LIN {X 0,Y 367.091,Z 171.622,A -85,B 0,C 180,E1 -12891.791,E2 -12891.791} C_VEL
LIN {X 0,Y 363.868,Z 162.966,A -85,B 0,C 180,E1 -12892.197,E2 -12892.197} C_VEL
LIN {X 0,Y 361.894,Z 153.404,A -85,B 0,C 180,E1 -12894.844,E2 -12894.844} C_VEL
LIN {X 0,Y 361.85,Z 153.414,A -85,B 0,C 180,E1 -12897.784,E2 -12897.784} C_VEL
LIN {X 0,Y 361.849,Z 153.41,A -85,B 0,C 180,E1 -12901.285,E2 -12901.285} C_VEL
LIN {X 0,Y 361.856,Z 153.408,A -85,B 0,C 180,E1 -12904.28,E2 -12904.28} C_VEL
LIN {X 0,Y 361.861,Z 153.409,A -85,B 0,C 180,E1 -12907.222,E2 -12907.222} C_VEL
LIN {X 0,Y 361.813,Z 153.413,A -85,B 0,C 180,E1 -12910.751,E2 -12910.751} C_VEL
LIN {X 0,Y 361.817,Z 153.412,A -85,B 0,C 180,E1 -12914.368,E2 -12914.368} C_VEL
LIN {X 0,Y 361.831,Z 153.414,A -85,B 0,C 180,E1 -12917.569,E2 -12917.569} C_VEL
LIN {X 0,Y 361.843,Z 153.411,A -85,B 0,C 180,E1 -12921.572,E2 -12921.572} C_VEL
LIN {X 0,Y 361.87,Z 153.407,A -85,B 0,C 180,E1 -12924.656,E2 -12924.656} C_VEL
LIN {X 0,Y 361.836,Z 153.411,A -85,B 0,C 180,E1 -12928.37,E2 -12928.37} C_VEL
LIN {X 0,Y 361.865,Z 153.412,A -85,B 0,C 180,E1 -12930.952,E2 -12930.952} C_VEL
LIN {X 0,Y 361.882,Z 153.409,A -85,B 0,C 180,E1 -12934.706,E2 -12934.706} C_VEL
LIN {X 0,Y 361.888,Z 153.406,A -85,B 0,C 180,E1 -12938.347,E2 -12938.347} C_VEL
LIN {X 0,Y 361.903,Z 153.403,A -85,B 0,C 180,E1 -12942.093,E2 -12942.093} C_VEL
LIN {X 0,Y 361.978,Z 153.394,A -85,B 0,C 180,E1 -12946.113,E2 -12946.113} C_VEL
LIN {X 0,Y 361.997,Z 153.392,A -85,B 0,C 180,E1 -12949.937,E2 -12949.937} C_VEL
LIN {X 0,Y 362.116,Z 153.374,A -85,B 0,C 180,E1 -12953.313,E2 -12953.313} C_VEL
LIN {X 0,Y 362.261,Z 153.359,A -85,B 0,C 180,E1 -12957.776,E2 -12957.776} C_VEL
LIN {X 0,Y 362.17,Z 153.368,A -85,B 0,C 180,E1 -12961.112,E2 -12961.112} C_VEL
LIN {X 0,Y 362.254,Z 153.361,A -85,B 0,C 180,E1 -12962.224,E2 -12962.224} C_VEL
LIN {X 0,Y 362.117,Z 153.375,A -85,B 0,C 180,E1 -12966.687,E2 -12966.687} C_VEL
LIN {X 0,Y 361.99,Z 153.394,A -85,B 0,C 180,E1 -12970.063,E2 -12970.063} C_VEL
LIN {X 0,Y 361.948,Z 153.4,A -85,B 0,C 180,E1 -12973.868,E2 -12973.868} C_VEL
LIN {X 0,Y 361.893,Z 153.405,A -85,B 0,C 180,E1 -12977.903,E2 -12977.903} C_VEL
LIN {X 0,Y 361.851,Z 153.412,A -85,B 0,C 180,E1 -12981.656,E2 -12981.656} C_VEL
LIN {X 0,Y 361.858,Z 153.413,A -85,B 0,C 180,E1 -12985.295,E2 -12985.295} C_VEL
LIN {X 0,Y 361.854,Z 153.412,A -85,B 0,C 180,E1 -12989.074,E2 -12989.074} C_VEL
LIN {X 0,Y 361.846,Z 153.413,A -85,B 0,C 180,E1 -12992.945,E2 -12992.945} C_VEL
LIN {X 0,Y 361.863,Z 153.408,A -85,B 0,C 180,E1 -12995.637,E2 -12995.637} C_VEL
LIN {X 0,Y 361.826,Z 153.417,A -85,B 0,C 180,E1 -12999.018,E2 -12999.018} C_VEL
LIN {X 0,Y 361.831,Z 153.416,A -85,B 0,C 180,E1 -13002.83,E2 -13002.83} C_VEL
LIN {X 0,Y 361.813,Z 153.413,A -85,B 0,C 180,E1 -13005.948,E2 -13005.948} C_VEL
LIN {X 0,Y 361.81,Z 153.414,A -85,B 0,C 180,E1 -13009.25,E2 -13009.25} C_VEL
LIN {X 0,Y 361.864,Z 153.408,A -85,B 0,C 180,E1 -13012.982,E2 -13012.982} C_VEL
LIN {X 0,Y 361.859,Z 153.412,A -85,B 0,C 180,E1 -13016.631,E2 -13016.631} C_VEL
LIN {X 0,Y 361.914,Z 153.447,A -85,B 0,C 180,E1 -13019.747,E2 -13019.747} C_VEL
LIN {X 0,Y 364.405,Z 165.157,A -85,B 0,C 180,E1 -13022.759,E2 -13022.759} C_VEL
LIN {X 0,Y 365.797,Z 172.397,A -85,B 0,C 180,E1 -13024.556,E2 -13024.556} C_VEL
LIN {X 0,Y 365.286,Z 179.494,A -85,B 0,C 180,E1 -13026.169,E2 -13026.169} C_VEL
LIN {X 0,Y 364.51,Z 187.222,A -85,B 0,C 180,E1 -13027.899,E2 -13027.899} C_VEL
LIN {X 0,Y 369.623,Z 218.201,A -85,B 0,C 180,E1 -13028.851,E2 -13028.851} C_VEL
LIN {X 0,Y 370.153,Z 223.288,A -85,B 0,C 180,E1 -13028.986,E2 -13028.986} C_VEL
LIN {X 0,Y 368.915,Z 295.915,A -85,B 0,C 180,E1 -13030.417,E2 -13030.417} C_VEL
LIN {X 0,Y 368.287,Z 309.127,A -85,B 0,C 180,E1 -13030.889,E2 -13030.889} C_VEL
LIN {X 0,Y 367.402,Z 321.258,A -85,B 0,C 180,E1 -13031.529,E2 -13031.529} C_VEL
LIN {X 0,Y 366.327,Z 333.507,A -85,B 0,C 180,E1 -13032.412,E2 -13032.412} C_VEL
LIN {X 0,Y 365.169,Z 345.099,A -85,B 0,C 180,E1 -13033.508,E2 -13033.508} C_VEL
LIN {X 0,Y 364.127,Z 355.365,A -85,B 0,C 180,E1 -13034.729,E2 -13034.729} C_VEL
LIN {X 0,Y 363.187,Z 364.085,A -85,B 0,C 180,E1 -13036.002,E2 -13036.002} C_VEL
LIN {X 0,Y 362.347,Z 371.969,A -85,B 0,C 180,E1 -13037.396,E2 -13037.396} C_VEL
LIN {X 0,Y 361.485,Z 379.671,A -85,B 0,C 180,E1 -13039.072,E2 -13039.072} C_VEL
LIN {X 0,Y 360.873,Z 386.781,A -85,B 0,C 180,E1 -13041.036,E2 -13041.036} C_VEL
LIN {X 0,Y 360.517,Z 391.513,A -85,B 0,C 180,E1 -13042.72,E2 -13042.72} C_VEL
LIN {X 0,Y 360.346,Z 395.131,A -85,B 0,C 180,E1 -13044.403,E2 -13044.403} C_VEL
LIN {X 0,Y 360.359,Z 397,A -85,B 0,C 180,E1 -13045.525,E2 -13045.525} C_VEL
LIN {X 0,Y 360.302,Z 398.399,A -85,B 0,C 180,E1 -13046.645,E2 -13046.645} C_VEL
LIN {X 0,Y 360.37,Z 400.012,A -85,B 0,C 180,E1 -13048.882,E2 -13048.882} C_VEL
LIN {X 0,Y 360.426,Z 400.229,A -85,B 0,C 180,E1 -13049.999,E2 -13049.999} C_VEL
LIN {X 0,Y 360.37,Z 400.007,A -85,B 0,C 180,E1 -13051.117,E2 -13051.117} C_VEL
LIN {X 0,Y 360.302,Z 398.391,A -85,B 0,C 180,E1 -13053.354,E2 -13053.354} C_VEL
LIN {X 0,Y 360.363,Z 396.988,A -85,B 0,C 180,E1 -13054.474,E2 -13054.474} C_VEL
LIN {X 0,Y 360.377,Z 394.412,A -85,B 0,C 180,E1 -13055.96,E2 -13055.96} C_VEL
LIN {X 0,Y 360.649,Z 390.046,A -85,B 0,C 180,E1 -13057.839,E2 -13057.839} C_VEL
LIN {X 0,Y 361.108,Z 383.913,A -85,B 0,C 180,E1 -13059.804,E2 -13059.804} C_VEL
LIN {X 0,Y 361.732,Z 377.218,A -85,B 0,C 180,E1 -13061.486,E2 -13061.486} C_VEL
LIN {X 0,Y 362.697,Z 368.92,A -85,B 0,C 180,E1 -13063.16,E2 -13063.16} C_VEL
LIN {X 0,Y 363.628,Z 360.414,A -85,B 0,C 180,E1 -13064.551,E2 -13064.551} C_VEL
LIN {X 0,Y 364.63,Z 349.903,A -85,B 0,C 180,E1 -13065.941,E2 -13065.941} C_VEL
LIN {X 0,Y 365.85,Z 338.082,A -85,B 0,C 180,E1 -13067.178,E2 -13067.178} C_VEL
LIN {X 0,Y 366.943,Z 326.189,A -85,B 0,C 180,E1 -13068.133,E2 -13068.133} C_VEL
LIN {X 0,Y 367.901,Z 313.816,A -85,B 0,C 180,E1 -13068.877,E2 -13068.877} C_VEL
LIN {X 0,Y 368.686,Z 301.1,A -85,B 0,C 180,E1 -13069.414,E2 -13069.414} C_VEL
LIN {X 0,Y 369.122,Z 287.728,A -85,B 0,C 180,E1 -13069.751,E2 -13069.751} C_VEL
LIN {X 0,Y 369.96,Z 220.882,A -85,B 0,C 180,E1 -13071.059,E2 -13071.059} C_VEL
LIN {X 0,Y 366.012,Z 195.478,A -85,B 0,C 180,E1 -13071.818,E2 -13071.818} C_VEL
LIN {X 0,Y 364.524,Z 187.205,A -85,B 0,C 180,E1 -13072.087,E2 -13072.087} C_VEL
LIN {X 0,Y 365.792,Z 174.22,A -85,B 0,C 180,E1 -13075.003,E2 -13075.003} C_VEL
LIN {X 0,Y 365.348,Z 169.998,A -85,B 0,C 180,E1 -13076.017,E2 -13076.017} C_VEL
LIN {X 0,Y 363.032,Z 158.382,A -85,B 0,C 180,E1 -13078.944,E2 -13078.944} C_VEL
LIN {X 0,Y 361.897,Z 153.408,A -85,B 0,C 180,E1 -13080.253,E2 -13080.253} C_VEL
LIN {X 0,Y 361.85,Z 153.408,A -85,B 0,C 180,E1 -13084.28,E2 -13084.28} C_VEL
LIN {X 0,Y 361.856,Z 153.411,A -85,B 0,C 180,E1 -13087.221,E2 -13087.221} C_VEL
LIN {X 0,Y 361.808,Z 153.414,A -85,B 0,C 180,E1 -13090.75,E2 -13090.75} C_VEL
LIN {X 0,Y 361.809,Z 153.413,A -85,B 0,C 180,E1 -13094.368,E2 -13094.368} C_VEL
LIN {X 0,Y 361.823,Z 153.414,A -85,B 0,C 180,E1 -13097.568,E2 -13097.568} C_VEL
LIN {X 0,Y 361.837,Z 153.411,A -85,B 0,C 180,E1 -13101.571,E2 -13101.571} C_VEL
LIN {X 0,Y 361.863,Z 153.41,A -85,B 0,C 180,E1 -13104.656,E2 -13104.656} C_VEL
LIN {X 0,Y 361.83,Z 153.412,A -85,B 0,C 180,E1 -13108.37,E2 -13108.37} C_VEL
LIN {X 0,Y 361.859,Z 153.411,A -85,B 0,C 180,E1 -13110.951,E2 -13110.951} C_VEL
LIN {X 0,Y 361.853,Z 153.414,A -85,B 0,C 180,E1 -13114.704,E2 -13114.704} C_VEL
LIN {X 0,Y 361.845,Z 153.412,A -85,B 0,C 180,E1 -13118.344,E2 -13118.344} C_VEL
LIN {X 0,Y 361.896,Z 153.405,A -85,B 0,C 180,E1 -13122.092,E2 -13122.092} C_VEL
LIN {X 0,Y 361.97,Z 153.397,A -85,B 0,C 180,E1 -13126.113,E2 -13126.113} C_VEL
LIN {X 0,Y 361.985,Z 153.394,A -85,B 0,C 180,E1 -13129.937,E2 -13129.937} C_VEL
LIN {X 0,Y 362.108,Z 153.376,A -85,B 0,C 180,E1 -13133.313,E2 -13133.313} C_VEL
LIN {X 0,Y 362.248,Z 153.362,A -85,B 0,C 180,E1 -13137.776,E2 -13137.776} C_VEL
LIN {X 0,Y 362.163,Z 153.369,A -85,B 0,C 180,E1 -13141.112,E2 -13141.112} C_VEL
LIN {X 0,Y 362.254,Z 153.361,A -85,B 0,C 180,E1 -13142.224,E2 -13142.224} C_VEL
LIN {X 0,Y 362.112,Z 153.375,A -85,B 0,C 180,E1 -13146.687,E2 -13146.687} C_VEL
LIN {X 0,Y 361.99,Z 153.393,A -85,B 0,C 180,E1 -13150.063,E2 -13150.063} C_VEL
LIN {X 0,Y 361.971,Z 153.396,A -85,B 0,C 180,E1 -13153.887,E2 -13153.887} C_VEL
LIN {X 0,Y 361.879,Z 153.405,A -85,B 0,C 180,E1 -13158.104,E2 -13158.104} C_VEL
LIN {X 0,Y 361.881,Z 153.407,A -85,B 0,C 180,E1 -13161.654,E2 -13161.654} C_VEL
LIN {X 0,Y 361.854,Z 153.413,A -85,B 0,C 180,E1 -13165.296,E2 -13165.296} C_VEL
LIN {X 0,Y 361.848,Z 153.414,A -85,B 0,C 180,E1 -13169.074,E2 -13169.074} C_VEL
LIN {X 0,Y 361.841,Z 153.414,A -85,B 0,C 180,E1 -13172.946,E2 -13172.946} C_VEL
LIN {X 0,Y 361.858,Z 153.408,A -85,B 0,C 180,E1 -13175.638,E2 -13175.638} C_VEL
LIN {X 0,Y 361.821,Z 153.416,A -85,B 0,C 180,E1 -13179.019,E2 -13179.019} C_VEL
LIN {X 0,Y 361.828,Z 153.417,A -85,B 0,C 180,E1 -13182.83,E2 -13182.83} C_VEL
LIN {X 0,Y 361.813,Z 153.413,A -85,B 0,C 180,E1 -13185.948,E2 -13185.948} C_VEL
LIN {X 0,Y 361.826,Z 153.412,A -85,B 0,C 180,E1 -13189.247,E2 -13189.247} C_VEL
LIN {X 0,Y 361.862,Z 153.408,A -85,B 0,C 180,E1 -13192.983,E2 -13192.983} C_VEL
LIN {X 0,Y 361.857,Z 153.411,A -85,B 0,C 180,E1 -13196.632,E2 -13196.632} C_VEL
LIN {X 0,Y 361.863,Z 153.407,A -85,B 0,C 180,E1 -13199.672,E2 -13199.672} C_VEL
LIN {X 0,Y 361.864,Z 153.406,A -85,B 0,C 180,E1 -13203.469,E2 -13203.469} C_VEL
LIN {X 0,Y 361.905,Z 153.596,A -85,B 0,C 180,E1 -13205.322,E2 -13205.322} C_VEL
LIN {X 0,Y 363.891,Z 162.985,A -85,B 0,C 180,E1 -13207.917,E2 -13207.917} C_VEL
LIN {X 0,Y 367.735,Z 173.936,A -85,B 0,C 180,E1 -13208.403,E2 -13208.403} C_VEL
LIN {X 0,Y 370.621,Z 188.653,A -85,B 0,C 180,E1 -13208.883,E2 -13208.883} C_VEL
LIN {X 0,Y 369.412,Z 265.31,A -85,B 0,C 180,E1 -13210.373,E2 -13210.373} C_VEL
LIN {X 0,Y 369.011,Z 278.206,A -85,B 0,C 180,E1 -13210.749,E2 -13210.749} C_VEL
LIN {X 0,Y 368.333,Z 291.445,A -85,B 0,C 180,E1 -13211.362,E2 -13211.362} C_VEL
LIN {X 0,Y 367.455,Z 303.827,A -85,B 0,C 180,E1 -13212.181,E2 -13212.181} C_VEL
LIN {X 0,Y 366.505,Z 314.918,A -85,B 0,C 180,E1 -13213.141,E2 -13213.141} C_VEL
LIN {X 0,Y 365.734,Z 324.837,A -85,B 0,C 180,E1 -13214.225,E2 -13214.225} C_VEL
LIN {X 0,Y 364.652,Z 334.372,A -85,B 0,C 180,E1 -13215.491,E2 -13215.491} C_VEL
LIN {X 0,Y 363.638,Z 342.859,A -85,B 0,C 180,E1 -13216.875,E2 -13216.875} C_VEL
LIN {X 0,Y 362.729,Z 351.099,A -85,B 0,C 180,E1 -13218.546,E2 -13218.546} C_VEL
LIN {X 0,Y 362.057,Z 356.737,A -85,B 0,C 180,E1 -13219.939,E2 -13219.939} C_VEL
LIN {X 0,Y 361.4,Z 362.232,A -85,B 0,C 180,E1 -13221.614,E2 -13221.614} C_VEL
LIN {X 0,Y 361.035,Z 366.54,A -85,B 0,C 180,E1 -13223.293,E2 -13223.293} C_VEL
LIN {X 0,Y 360.844,Z 368.819,A -85,B 0,C 180,E1 -13224.412,E2 -13224.412} C_VEL
LIN {X 0,Y 360.627,Z 370.676,A -85,B 0,C 180,E1 -13225.53,E2 -13225.53} C_VEL
LIN {X 0,Y 360.515,Z 372.072,A -85,B 0,C 180,E1 -13226.648,E2 -13226.648} C_VEL
LIN {X 0,Y 360.424,Z 373.675,A -85,B 0,C 180,E1 -13228.883,E2 -13228.883} C_VEL
LIN {X 0,Y 360.429,Z 373.906,A -85,B 0,C 180,E1 -13230.001,E2 -13230.001} C_VEL
LIN {X 0,Y 360.424,Z 373.718,A -85,B 0,C 180,E1 -13231.118,E2 -13231.118} C_VEL
LIN {X 0,Y 360.51,Z 372.171,A -85,B 0,C 180,E1 -13233.353,E2 -13233.353} C_VEL
LIN {X 0,Y 360.619,Z 370.818,A -85,B 0,C 180,E1 -13234.472,E2 -13234.472} C_VEL
LIN {X 0,Y 360.934,Z 367.955,A -85,B 0,C 180,E1 -13236.148,E2 -13236.148} C_VEL
LIN {X 0,Y 361.212,Z 364.08,A -85,B 0,C 180,E1 -13237.828,E2 -13237.828} C_VEL
LIN {X 0,Y 361.778,Z 359.072,A -85,B 0,C 180,E1 -13239.505,E2 -13239.505} C_VEL
LIN {X 0,Y 362.531,Z 352.766,A -85,B 0,C 180,E1 -13241.179,E2 -13241.179} C_VEL
LIN {X 0,Y 363.433,Z 344.872,A -85,B 0,C 180,E1 -13242.85,E2 -13242.85} C_VEL
LIN {X 0,Y 364.45,Z 336.819,A -85,B 0,C 180,E1 -13244.234,E2 -13244.234} C_VEL
LIN {X 0,Y 365.523,Z 326.991,A -85,B 0,C 180,E1 -13245.616,E2 -13245.616} C_VEL
LIN {X 0,Y 366.352,Z 317.324,A -85,B 0,C 180,E1 -13246.724,E2 -13246.724} C_VEL
LIN {X 0,Y 367.287,Z 306.852,A -85,B 0,C 180,E1 -13247.684,E2 -13247.684} C_VEL
LIN {X 0,Y 368.181,Z 294.238,A -85,B 0,C 180,E1 -13248.575,E2 -13248.575} C_VEL
LIN {X 0,Y 368.908,Z 281.603,A -85,B 0,C 180,E1 -13249.222,E2 -13249.222} C_VEL
LIN {X 0,Y 369.266,Z 273.016,A -85,B 0,C 180,E1 -13249.53,E2 -13249.53} C_VEL
LIN {X 0,Y 368.777,Z 267.258,A -85,B 0,C 180,E1 -13249.725,E2 -13249.725} C_VEL
LIN {X 0,Y 363.714,Z 248.579,A -85,B 0,C 180,E1 -13250.412,E2 -13250.412} C_VEL
LIN {X 0,Y 363.144,Z 242.768,A -85,B 0,C 180,E1 -13250.561,E2 -13250.561} C_VEL
LIN {X 0,Y 363.993,Z 188.874,A -85,B 0,C 180,E1 -13251.629,E2 -13251.629} C_VEL
LIN {X 0,Y 360.675,Z 173.698,A -85,B 0,C 180,E1 -13252.16,E2 -13252.16} C_VEL
LIN {X 0,Y 356.72,Z 163.234,A -85,B 0,C 180,E1 -13252.667,E2 -13252.667} C_VEL
LIN {X 0,Y 354.855,Z 154.281,A -85,B 0,C 180,E1 -13255.202,E2 -13255.202} C_VEL
LIN {X 0,Y 354.804,Z 154.288,A -85,B 0,C 180,E1 -13258.385,E2 -13258.385} C_VEL
LIN {X 0,Y 354.789,Z 154.289,A -85,B 0,C 180,E1 -13262.333,E2 -13262.333} C_VEL
LIN {X 0,Y 354.823,Z 154.289,A -85,B 0,C 180,E1 -13265.699,E2 -13265.699} C_VEL
LIN {X 0,Y 354.769,Z 154.295,A -85,B 0,C 180,E1 -13269.412,E2 -13269.412} C_VEL
LIN {X 0,Y 354.786,Z 154.289,A -85,B 0,C 180,E1 -13272.867,E2 -13272.867} C_VEL
LIN {X 0,Y 354.767,Z 154.29,A -85,B 0,C 180,E1 -13276.103,E2 -13276.103} C_VEL
LIN {X 0,Y 354.766,Z 154.296,A -85,B 0,C 180,E1 -13279.176,E2 -13279.176} C_VEL
LIN {X 0,Y 354.799,Z 154.287,A -85,B 0,C 180,E1 -13282.404,E2 -13282.404} C_VEL
LIN {X 0,Y 354.808,Z 154.29,A -85,B 0,C 180,E1 -13284.94,E2 -13284.94} C_VEL
LIN {X 0,Y 354.792,Z 154.288,A -85,B 0,C 180,E1 -13288.405,E2 -13288.405} C_VEL
LIN {X 0,Y 354.799,Z 154.286,A -85,B 0,C 180,E1 -13291.614,E2 -13291.614} C_VEL
LIN {X 0,Y 354.834,Z 154.282,A -85,B 0,C 180,E1 -13295.657,E2 -13295.657} C_VEL
LIN {X 0,Y 354.834,Z 154.284,A -85,B 0,C 180,E1 -13299.113,E2 -13299.113} C_VEL
LIN {X 0,Y 354.85,Z 154.284,A -85,B 0,C 180,E1 -13302.717,E2 -13302.717} C_VEL
LIN {X 0,Y 354.938,Z 154.272,A -85,B 0,C 180,E1 -13306.254,E2 -13306.254} C_VEL
LIN {X 0,Y 354.953,Z 154.268,A -85,B 0,C 180,E1 -13309.735,E2 -13309.735} C_VEL
LIN {X 0,Y 355.082,Z 154.25,A -85,B 0,C 180,E1 -13313.18,E2 -13313.18} C_VEL
LIN {X 0,Y 355.223,Z 154.236,A -85,B 0,C 180,E1 -13317.732,E2 -13317.732} C_VEL
LIN {X 0,Y 355.142,Z 154.242,A -85,B 0,C 180,E1 -13321.134,E2 -13321.134} C_VEL
LIN {X 0,Y 355.216,Z 154.237,A -85,B 0,C 180,E1 -13322.268,E2 -13322.268} C_VEL
LIN {X 0,Y 355.083,Z 154.251,A -85,B 0,C 180,E1 -13326.82,E2 -13326.82} C_VEL
LIN {X 0,Y 354.946,Z 154.269,A -85,B 0,C 180,E1 -13330.265,E2 -13330.265} C_VEL
LIN {X 0,Y 354.89,Z 154.278,A -85,B 0,C 180,E1 -13333.985,E2 -13333.985} C_VEL
LIN {X 0,Y 354.833,Z 154.283,A -85,B 0,C 180,E1 -13338.065,E2 -13338.065} C_VEL
LIN {X 0,Y 354.803,Z 154.286,A -85,B 0,C 180,E1 -13342.108,E2 -13342.108} C_VEL
LIN {X 0,Y 354.797,Z 154.288,A -85,B 0,C 180,E1 -13345.835,E2 -13345.835} C_VEL
LIN {X 0,Y 354.791,Z 154.289,A -85,B 0,C 180,E1 -13349.684,E2 -13349.684} C_VEL
LIN {X 0,Y 354.785,Z 154.288,A -85,B 0,C 180,E1 -13352.334,E2 -13352.334} C_VEL
LIN {X 0,Y 354.817,Z 154.285,A -85,B 0,C 180,E1 -13355.698,E2 -13355.698} C_VEL
LIN {X 0,Y 354.768,Z 154.292,A -85,B 0,C 180,E1 -13359.413,E2 -13359.413} C_VEL
LIN {X 0,Y 354.784,Z 154.295,A -85,B 0,C 180,E1 -13362.866,E2 -13362.866} C_VEL
LIN {X 0,Y 354.762,Z 154.292,A -85,B 0,C 180,E1 -13366.103,E2 -13366.103} C_VEL
LIN {X 0,Y 354.763,Z 154.292,A -85,B 0,C 180,E1 -13369.176,E2 -13369.176} C_VEL
LIN {X 0,Y 354.801,Z 154.29,A -85,B 0,C 180,E1 -13372.404,E2 -13372.404} C_VEL
LIN {X 0,Y 354.812,Z 154.288,A -85,B 0,C 180,E1 -13374.941,E2 -13374.941} C_VEL
LIN {X 0,Y 354.794,Z 154.293,A -85,B 0,C 180,E1 -13378.405,E2 -13378.405} C_VEL
LIN {X 0,Y 354.862,Z 154.356,A -85,B 0,C 180,E1 -13379.379,E2 -13379.379} C_VEL
LIN {X 0,Y 357.269,Z 165.329,A -85,B 0,C 180,E1 -13382.278,E2 -13382.278} C_VEL
LIN {X 0,Y 358.884,Z 174.019,A -85,B 0,C 180,E1 -13384.48,E2 -13384.48} C_VEL
LIN {X 0,Y 358.14,Z 183.133,A -85,B 0,C 180,E1 -13386.585,E2 -13386.585} C_VEL
LIN {X 0,Y 357.664,Z 186.937,A -85,B 0,C 180,E1 -13387.449,E2 -13387.449} C_VEL
LIN {X 0,Y 362.658,Z 216.507,A -85,B 0,C 180,E1 -13388.395,E2 -13388.395} C_VEL
LIN {X 0,Y 363.534,Z 223.627,A -85,B 0,C 180,E1 -13388.597,E2 -13388.597} C_VEL
LIN {X 0,Y 362.248,Z 295.669,A -85,B 0,C 180,E1 -13390.041,E2 -13390.041} C_VEL
LIN {X 0,Y 361.592,Z 308.877,A -85,B 0,C 180,E1 -13390.521,E2 -13390.521} C_VEL
LIN {X 0,Y 360.677,Z 321.006,A -85,B 0,C 180,E1 -13391.172,E2 -13391.172} C_VEL
LIN {X 0,Y 359.573,Z 333.252,A -85,B 0,C 180,E1 -13392.071,E2 -13392.071} C_VEL
LIN {X 0,Y 358.335,Z 344.842,A -85,B 0,C 180,E1 -13393.184,E2 -13393.184} C_VEL
LIN {X 0,Y 357.18,Z 355.873,A -85,B 0,C 180,E1 -13394.53,E2 -13394.53} C_VEL
LIN {X 0,Y 356.091,Z 365.505,A -85,B 0,C 180,E1 -13396.008,E2 -13396.008} C_VEL
LIN {X 0,Y 355.061,Z 374.452,A -85,B 0,C 180,E1 -13397.714,E2 -13397.714} C_VEL
LIN {X 0,Y 354.286,Z 381.656,A -85,B 0,C 180,E1 -13399.426,E2 -13399.426} C_VEL
LIN {X 0,Y 353.691,Z 388.222,A -85,B 0,C 180,E1 -13401.429,E2 -13401.429} C_VEL
LIN {X 0,Y 353.397,Z 392.569,A -85,B 0,C 180,E1 -13403.147,E2 -13403.147} C_VEL
LIN {X 0,Y 353.282,Z 394.873,A -85,B 0,C 180,E1 -13404.291,E2 -13404.291} C_VEL
LIN {X 0,Y 353.269,Z 396.741,A -85,B 0,C 180,E1 -13405.435,E2 -13405.435} C_VEL
LIN {X 0,Y 353.223,Z 398.141,A -85,B 0,C 180,E1 -13406.577,E2 -13406.577} C_VEL
LIN {X 0,Y 353.271,Z 399.753,A -85,B 0,C 180,E1 -13408.859,E2 -13408.859} C_VEL
LIN {X 0,Y 353.331,Z 399.97,A -85,B 0,C 180,E1 -13409.999,E2 -13409.999} C_VEL
LIN {X 0,Y 353.271,Z 399.748,A -85,B 0,C 180,E1 -13411.139,E2 -13411.139} C_VEL
LIN {X 0,Y 353.224,Z 398.132,A -85,B 0,C 180,E1 -13413.421,E2 -13413.421} C_VEL
LIN {X 0,Y 353.274,Z 396.728,A -85,B 0,C 180,E1 -13414.563,E2 -13414.563} C_VEL
LIN {X 0,Y 353.275,Z 394.483,A -85,B 0,C 180,E1 -13415.904,E2 -13415.904} C_VEL
LIN {X 0,Y 353.574,Z 389.784,A -85,B 0,C 180,E1 -13417.997,E2 -13417.997} C_VEL
LIN {X 0,Y 354.073,Z 383.651,A -85,B 0,C 180,E1 -13420.001,E2 -13420.001} C_VEL
LIN {X 0,Y 354.719,Z 376.955,A -85,B 0,C 180,E1 -13421.716,E2 -13421.716} C_VEL
LIN {X 0,Y 355.754,Z 368.658,A -85,B 0,C 180,E1 -13423.421,E2 -13423.421} C_VEL
LIN {X 0,Y 356.746,Z 360.152,A -85,B 0,C 180,E1 -13424.838,E2 -13424.838} C_VEL
LIN {X 0,Y 357.763,Z 349.639,A -85,B 0,C 180,E1 -13426.255,E2 -13426.255} C_VEL
LIN {X 0,Y 359.054,Z 337.818,A -85,B 0,C 180,E1 -13427.513,E2 -13427.513} C_VEL
LIN {X 0,Y 360.175,Z 325.923,A -85,B 0,C 180,E1 -13428.486,E2 -13428.486} C_VEL
LIN {X 0,Y 361.195,Z 313.549,A -85,B 0,C 180,E1 -13429.241,E2 -13429.241} C_VEL
LIN {X 0,Y 362.001,Z 300.83,A -85,B 0,C 180,E1 -13429.787,E2 -13429.787} C_VEL
LIN {X 0,Y 362.456,Z 287.449,A -85,B 0,C 180,E1 -13430.13,E2 -13430.13} C_VEL
LIN {X 0,Y 363.351,Z 221.934,A -85,B 0,C 180,E1 -13431.433,E2 -13431.433} C_VEL
LIN {X 0,Y 359.5,Z 196.978,A -85,B 0,C 180,E1 -13432.197,E2 -13432.197} C_VEL
LIN {X 0,Y 357.695,Z 186.921,A -85,B 0,C 180,E1 -13432.536,E2 -13432.536} C_VEL
LIN {X 0,Y 358.877,Z 175.254,A -85,B 0,C 180,E1 -13435.209,E2 -13435.209} C_VEL
LIN {X 0,Y 358.144,Z 169.993,A -85,B 0,C 180,E1 -13436.514,E2 -13436.514} C_VEL
LIN {X 0,Y 355.842,Z 158.873,A -85,B 0,C 180,E1 -13439.394,E2 -13439.394} C_VEL
LIN {X 0,Y 354.831,Z 154.288,A -85,B 0,C 180,E1 -13440.664,E2 -13440.664} C_VEL
LIN {X 0,Y 354.803,Z 154.29,A -85,B 0,C 180,E1 -13443.701,E2 -13443.701} C_VEL
LIN {X 0,Y 354.791,Z 154.287,A -85,B 0,C 180,E1 -13446.459,E2 -13446.459} C_VEL
LIN {X 0,Y 354.764,Z 154.296,A -85,B 0,C 180,E1 -13449.411,E2 -13449.411} C_VEL
LIN {X 0,Y 354.78,Z 154.291,A -85,B 0,C 180,E1 -13452.866,E2 -13452.866} C_VEL
LIN {X 0,Y 354.757,Z 154.292,A -85,B 0,C 180,E1 -13456.102,E2 -13456.102} C_VEL
LIN {X 0,Y 354.76,Z 154.297,A -85,B 0,C 180,E1 -13459.175,E2 -13459.175} C_VEL
LIN {X 0,Y 354.793,Z 154.288,A -85,B 0,C 180,E1 -13462.403,E2 -13462.403} C_VEL
LIN {X 0,Y 354.802,Z 154.292,A -85,B 0,C 180,E1 -13464.94,E2 -13464.94} C_VEL
LIN {X 0,Y 354.786,Z 154.29,A -85,B 0,C 180,E1 -13468.405,E2 -13468.405} C_VEL
LIN {X 0,Y 354.791,Z 154.287,A -85,B 0,C 180,E1 -13471.614,E2 -13471.614} C_VEL
LIN {X 0,Y 354.796,Z 154.287,A -85,B 0,C 180,E1 -13475.419,E2 -13475.419} C_VEL
LIN {X 0,Y 354.812,Z 154.286,A -85,B 0,C 180,E1 -13479.112,E2 -13479.112} C_VEL
LIN {X 0,Y 354.842,Z 154.283,A -85,B 0,C 180,E1 -13482.717,E2 -13482.717} C_VEL
LIN {X 0,Y 354.93,Z 154.275,A -85,B 0,C 180,E1 -13486.254,E2 -13486.254} C_VEL
LIN {X 0,Y 354.941,Z 154.27,A -85,B 0,C 180,E1 -13489.735,E2 -13489.735} C_VEL
LIN {X 0,Y 355.074,Z 154.252,A -85,B 0,C 180,E1 -13493.18,E2 -13493.18} C_VEL
LIN {X 0,Y 355.209,Z 154.237,A -85,B 0,C 180,E1 -13497.732,E2 -13497.732} C_VEL
LIN {X 0,Y 355.135,Z 154.245,A -85,B 0,C 180,E1 -13501.134,E2 -13501.134} C_VEL
LIN {X 0,Y 355.216,Z 154.237,A -85,B 0,C 180,E1 -13502.268,E2 -13502.268} C_VEL
LIN {X 0,Y 355.078,Z 154.251,A -85,B 0,C 180,E1 -13506.82,E2 -13506.82} C_VEL
LIN {X 0,Y 354.947,Z 154.269,A -85,B 0,C 180,E1 -13510.265,E2 -13510.265} C_VEL
LIN {X 0,Y 354.914,Z 154.274,A -85,B 0,C 180,E1 -13514.006,E2 -13514.006} C_VEL
LIN {X 0,Y 354.836,Z 154.282,A -85,B 0,C 180,E1 -13518.07,E2 -13518.07} C_VEL
LIN {X 0,Y 354.821,Z 154.284,A -85,B 0,C 180,E1 -13522.107,E2 -13522.107} C_VEL
LIN {X 0,Y 354.796,Z 154.287,A -85,B 0,C 180,E1 -13525.836,E2 -13525.836} C_VEL
LIN {X 0,Y 354.789,Z 154.289,A -85,B 0,C 180,E1 -13529.685,E2 -13529.685} C_VEL
LIN {X 0,Y 354.779,Z 154.289,A -85,B 0,C 180,E1 -13532.334,E2 -13532.334} C_VEL
LIN {X 0,Y 354.812,Z 154.285,A -85,B 0,C 180,E1 -13535.699,E2 -13535.699} C_VEL
LIN {X 0,Y 354.762,Z 154.292,A -85,B 0,C 180,E1 -13539.413,E2 -13539.413} C_VEL
LIN {X 0,Y 354.78,Z 154.294,A -85,B 0,C 180,E1 -13542.868,E2 -13542.868} C_VEL
LIN {X 0,Y 354.762,Z 154.292,A -85,B 0,C 180,E1 -13546.105,E2 -13546.105} C_VEL
LIN {X 0,Y 354.778,Z 154.29,A -85,B 0,C 180,E1 -13549.179,E2 -13549.179} C_VEL
LIN {X 0,Y 354.798,Z 154.291,A -85,B 0,C 180,E1 -13552.405,E2 -13552.405} C_VEL
LIN {X 0,Y 354.809,Z 154.287,A -85,B 0,C 180,E1 -13554.942,E2 -13554.942} C_VEL
LIN {X 0,Y 354.792,Z 154.293,A -85,B 0,C 180,E1 -13558.406,E2 -13558.406} C_VEL
LIN {X 0,Y 354.799,Z 154.287,A -85,B 0,C 180,E1 -13561.616,E2 -13561.616} C_VEL
LIN {X 0,Y 354.865,Z 154.436,A -85,B 0,C 180,E1 -13564.956,E2 -13564.956} C_VEL
LIN {X 0,Y 356.718,Z 163.241,A -85,B 0,C 180,E1 -13567.444,E2 -13567.444} C_VEL
LIN {X 0,Y 361.308,Z 175.825,A -85,B 0,C 180,E1 -13568.033,E2 -13568.033} C_VEL
LIN {X 0,Y 364.003,Z 188.937,A -85,B 0,C 180,E1 -13568.48,E2 -13568.48} C_VEL
LIN {X 0,Y 362.737,Z 265.591,A -85,B 0,C 180,E1 -13569.997,E2 -13569.997} C_VEL
LIN {X 0,Y 362.34,Z 278.477,A -85,B 0,C 180,E1 -13570.38,E2 -13570.38} C_VEL
LIN {X 0,Y 361.627,Z 291.712,A -85,B 0,C 180,E1 -13571.003,E2 -13571.003} C_VEL
LIN {X 0,Y 360.724,Z 304.091,A -85,B 0,C 180,E1 -13571.837,E2 -13571.837} C_VEL
LIN {X 0,Y 359.712,Z 315.182,A -85,B 0,C 180,E1 -13572.813,E2 -13572.813} C_VEL
LIN {X 0,Y 358.885,Z 325.393,A -85,B 0,C 180,E1 -13573.952,E2 -13573.952} C_VEL
LIN {X 0,Y 357.794,Z 334.634,A -85,B 0,C 180,E1 -13575.206,E2 -13575.206} C_VEL
LIN {X 0,Y 356.73,Z 343.121,A -85,B 0,C 180,E1 -13576.616,E2 -13576.616} C_VEL
LIN {X 0,Y 355.757,Z 351.361,A -85,B 0,C 180,E1 -13578.318,E2 -13578.318} C_VEL
LIN {X 0,Y 355.055,Z 356.999,A -85,B 0,C 180,E1 -13579.739,E2 -13579.739} C_VEL
LIN {X 0,Y 354.382,Z 362.492,A -85,B 0,C 180,E1 -13581.447,E2 -13581.447} C_VEL
LIN {X 0,Y 353.908,Z 367.565,A -85,B 0,C 180,E1 -13583.513,E2 -13583.513} C_VEL
LIN {X 0,Y 353.565,Z 370.936,A -85,B 0,C 180,E1 -13585.44,E2 -13585.44} C_VEL
LIN {X 0,Y 353.431,Z 372.332,A -85,B 0,C 180,E1 -13586.581,E2 -13586.581} C_VEL
LIN {X 0,Y 353.33,Z 373.934,A -85,B 0,C 180,E1 -13588.861,E2 -13588.861} C_VEL
LIN {X 0,Y 353.334,Z 374.165,A -85,B 0,C 180,E1 -13590.001,E2 -13590.001} C_VEL
LIN {X 0,Y 353.329,Z 373.977,A -85,B 0,C 180,E1 -13591.14,E2 -13591.14} C_VEL
LIN {X 0,Y 353.426,Z 372.429,A -85,B 0,C 180,E1 -13593.421,E2 -13593.421} C_VEL
LIN {X 0,Y 353.559,Z 371.076,A -85,B 0,C 180,E1 -13594.561,E2 -13594.561} C_VEL
LIN {X 0,Y 353.919,Z 367.823,A -85,B 0,C 180,E1 -13596.47,E2 -13596.47} C_VEL
LIN {X 0,Y 354.323,Z 362.784,A -85,B 0,C 180,E1 -13598.556,E2 -13598.556} C_VEL
LIN {X 0,Y 355.191,Z 356.354,A -85,B 0,C 180,E1 -13600.546,E2 -13600.546} C_VEL
LIN {X 0,Y 356.021,Z 349.291,A -85,B 0,C 180,E1 -13602.252,E2 -13602.252} C_VEL
LIN {X 0,Y 357.093,Z 340.486,A -85,B 0,C 180,E1 -13603.952,E2 -13603.952} C_VEL
LIN {X 0,Y 358.232,Z 331.445,A -85,B 0,C 180,E1 -13605.358,E2 -13605.358} C_VEL
LIN {X 0,Y 359.275,Z 320.737,A -85,B 0,C 180,E1 -13606.704,E2 -13606.704} C_VEL
LIN {X 0,Y 360.261,Z 310.298,A -85,B 0,C 180,E1 -13607.747,E2 -13607.747} C_VEL
LIN {X 0,Y 361.128,Z 299.771,A -85,B 0,C 180,E1 -13608.583,E2 -13608.583} C_VEL
LIN {X 0,Y 361.933,Z 287.088,A -85,B 0,C 180,E1 -13609.349,E2 -13609.349} C_VEL
LIN {X 0,Y 362.565,Z 274.459,A -85,B 0,C 180,E1 -13609.867,E2 -13609.867} C_VEL
LIN {X 0,Y 363.042,Z 256.539,A -85,B 0,C 180,E1 -13610.282,E2 -13610.282} C_VEL
LIN {X 0,Y 363.144,Z 242.768,A -85,B 0,C 180,E1 -13610.561,E2 -13610.561} C_VEL
LIN {X 0,Y 362.583,Z 236.96,A -85,B 0,C 180,E1 -13610.716,E2 -13610.716} C_VEL
LIN {X 0,Y 357.622,Z 218.257,A -85,B 0,C 180,E1 -13611.415,E2 -13611.415} C_VEL
LIN {X 0,Y 357.129,Z 212.448,A -85,B 0,C 180,E1 -13611.57,E2 -13611.57} C_VEL
LIN {X 0,Y 357.414,Z 189.999,A -85,B 0,C 180,E1 -13612.028,E2 -13612.028} C_VEL
LIN {X 0,Y 354.443,Z 176.272,A -85,B 0,C 180,E1 -13612.52,E2 -13612.52} C_VEL
LIN {X 0,Y 349.572,Z 163.504,A -85,B 0,C 180,E1 -13613.157,E2 -13613.157} C_VEL
LIN {X 0,Y 347.806,Z 155.161,A -85,B 0,C 180,E1 -13615.59,E2 -13615.59} C_VEL
LIN {X 0,Y 347.757,Z 155.169,A -85,B 0,C 180,E1 -13619.656,E2 -13619.656} C_VEL
LIN {X 0,Y 347.744,Z 155.166,A -85,B 0,C 180,E1 -13623.071,E2 -13623.071} C_VEL
LIN {X 0,Y 347.771,Z 155.164,A -85,B 0,C 180,E1 -13626.065,E2 -13626.065} C_VEL
LIN {X 0,Y 347.732,Z 155.167,A -85,B 0,C 180,E1 -13628.795,E2 -13628.795} C_VEL
LIN {X 0,Y 347.745,Z 155.168,A -85,B 0,C 180,E1 -13631.831,E2 -13631.831} C_VEL
LIN {X 0,Y 347.706,Z 155.173,A -85,B 0,C 180,E1 -13635.027,E2 -13635.027} C_VEL
LIN {X 0,Y 347.742,Z 155.166,A -85,B 0,C 180,E1 -13638.399,E2 -13638.399} C_VEL
LIN {X 0,Y 347.755,Z 155.166,A -85,B 0,C 180,E1 -13642.678,E2 -13642.678} C_VEL
LIN {X 0,Y 347.748,Z 155.164,A -85,B 0,C 180,E1 -13645.956,E2 -13645.956} C_VEL
LIN {X 0,Y 347.738,Z 155.166,A -85,B 0,C 180,E1 -13649.651,E2 -13649.651} C_VEL
LIN {X 0,Y 347.748,Z 155.165,A -85,B 0,C 180,E1 -13653.601,E2 -13653.601} C_VEL
LIN {X 0,Y 347.769,Z 155.163,A -85,B 0,C 180,E1 -13656.16,E2 -13656.16} C_VEL
LIN {X 0,Y 347.78,Z 155.161,A -85,B 0,C 180,E1 -13659.907,E2 -13659.907} C_VEL
LIN {X 0,Y 347.795,Z 155.158,A -85,B 0,C 180,E1 -13663.566,E2 -13663.566} C_VEL
LIN {X 0,Y 347.885,Z 155.148,A -85,B 0,C 180,E1 -13667.16,E2 -13667.16} C_VEL
LIN {X 0,Y 347.933,Z 155.143,A -85,B 0,C 180,E1 -13670.7,E2 -13670.7} C_VEL
LIN {X 0,Y 348.033,Z 155.133,A -85,B 0,C 180,E1 -13674.205,E2 -13674.205} C_VEL
LIN {X 0,Y 348.184,Z 155.112,A -85,B 0,C 180,E1 -13677.686,E2 -13677.686} C_VEL
LIN {X 0,Y 348.113,Z 155.117,A -85,B 0,C 180,E1 -13681.157,E2 -13681.157} C_VEL
LIN {X 0,Y 348.177,Z 155.113,A -85,B 0,C 180,E1 -13682.314,E2 -13682.314} C_VEL
LIN {X 0,Y 348.051,Z 155.127,A -85,B 0,C 180,E1 -13686.959,E2 -13686.959} C_VEL
LIN {X 0,Y 347.885,Z 155.147,A -85,B 0,C 180,E1 -13690.476,E2 -13690.476} C_VEL
LIN {X 0,Y 347.85,Z 155.153,A -85,B 0,C 180,E1 -13694.119,E2 -13694.119} C_VEL
LIN {X 0,Y 347.786,Z 155.16,A -85,B 0,C 180,E1 -13698.238,E2 -13698.238} C_VEL
LIN {X 0,Y 347.761,Z 155.166,A -85,B 0,C 180,E1 -13701.624,E2 -13701.624} C_VEL
LIN {X 0,Y 347.735,Z 155.169,A -85,B 0,C 180,E1 -13705.114,E2 -13705.114} C_VEL
LIN {X 0,Y 347.723,Z 155.169,A -85,B 0,C 180,E1 -13707.702,E2 -13707.702} C_VEL
LIN {X 0,Y 347.734,Z 155.166,A -85,B 0,C 180,E1 -13710.349,E2 -13710.349} C_VEL
LIN {X 0,Y 347.747,Z 155.164,A -85,B 0,C 180,E1 -13714.044,E2 -13714.044} C_VEL
LIN {X 0,Y 347.755,Z 155.166,A -85,B 0,C 180,E1 -13717.322,E2 -13717.322} C_VEL
LIN {X 0,Y 347.741,Z 155.166,A -85,B 0,C 180,E1 -13721.601,E2 -13721.601} C_VEL
LIN {X 0,Y 347.701,Z 155.174,A -85,B 0,C 180,E1 -13725.028,E2 -13725.028} C_VEL
LIN {X 0,Y 347.738,Z 155.169,A -85,B 0,C 180,E1 -13728.4,E2 -13728.4} C_VEL
LIN {X 0,Y 347.757,Z 155.169,A -85,B 0,C 180,E1 -13732.678,E2 -13732.678} C_VEL
LIN {X 0,Y 347.749,Z 155.167,A -85,B 0,C 180,E1 -13735.956,E2 -13735.956} C_VEL
LIN {X 0,Y 347.778,Z 155.221,A -85,B 0,C 180,E1 -13738.982,E2 -13738.982} C_VEL
LIN {X 0,Y 350.418,Z 167.094,A -85,B 0,C 180,E1 -13742.194,E2 -13742.194} C_VEL
LIN {X 0,Y 351.997,Z 176.388,A -85,B 0,C 180,E1 -13744.584,E2 -13744.584} C_VEL
LIN {X 0,Y 350.886,Z 186.654,A -85,B 0,C 180,E1 -13746.984,E2 -13746.984} C_VEL
LIN {X 0,Y 355.915,Z 216.263,A -85,B 0,C 180,E1 -13747.964,E2 -13747.964} C_VEL
LIN {X 0,Y 356.912,Z 224.696,A -85,B 0,C 180,E1 -13748.207,E2 -13748.207} C_VEL
LIN {X 0,Y 355.591,Z 295.423,A -85,B 0,C 180,E1 -13749.651,E2 -13749.651} C_VEL
LIN {X 0,Y 354.92,Z 308.626,A -85,B 0,C 180,E1 -13750.14,E2 -13750.14} C_VEL
LIN {X 0,Y 353.962,Z 320.753,A -85,B 0,C 180,E1 -13750.801,E2 -13750.801} C_VEL
LIN {X 0,Y 352.812,Z 332.997,A -85,B 0,C 180,E1 -13751.715,E2 -13751.715} C_VEL
LIN {X 0,Y 351.521,Z 344.585,A -85,B 0,C 180,E1 -13752.848,E2 -13752.848} C_VEL
LIN {X 0,Y 350.336,Z 355.033,A -85,B 0,C 180,E1 -13754.138,E2 -13754.138} C_VEL
LIN {X 0,Y 349.384,Z 363.57,A -85,B 0,C 180,E1 -13755.437,E2 -13755.437} C_VEL
LIN {X 0,Y 348.45,Z 371.453,A -85,B 0,C 180,E1 -13756.885,E2 -13756.885} C_VEL
LIN {X 0,Y 347.458,Z 379.152,A -85,B 0,C 180,E1 -13758.626,E2 -13758.626} C_VEL
LIN {X 0,Y 346.781,Z 386.263,A -85,B 0,C 180,E1 -13760.669,E2 -13760.669} C_VEL
LIN {X 0,Y 346.391,Z 390.995,A -85,B 0,C 180,E1 -13762.421,E2 -13762.421} C_VEL
LIN {X 0,Y 346.201,Z 394.614,A -85,B 0,C 180,E1 -13764.174,E2 -13764.174} C_VEL
LIN {X 0,Y 346.166,Z 396.482,A -85,B 0,C 180,E1 -13765.341,E2 -13765.341} C_VEL
LIN {X 0,Y 346.147,Z 397.882,A -85,B 0,C 180,E1 -13766.507,E2 -13766.507} C_VEL
LIN {X 0,Y 346.172,Z 399.493,A -85,B 0,C 180,E1 -13768.836,E2 -13768.836} C_VEL
LIN {X 0,Y 346.235,Z 399.711,A -85,B 0,C 180,E1 -13769.999,E2 -13769.999} C_VEL
LIN {X 0,Y 346.171,Z 399.488,A -85,B 0,C 180,E1 -13771.163,E2 -13771.163} C_VEL
LIN {X 0,Y 346.147,Z 397.873,A -85,B 0,C 180,E1 -13773.491,E2 -13773.491} C_VEL
LIN {X 0,Y 346.17,Z 396.467,A -85,B 0,C 180,E1 -13774.657,E2 -13774.657} C_VEL
LIN {X 0,Y 346.239,Z 393.515,A -85,B 0,C 180,E1 -13776.409,E2 -13776.409} C_VEL
LIN {X 0,Y 346.52,Z 389.523,A -85,B 0,C 180,E1 -13778.161,E2 -13778.161} C_VEL
LIN {X 0,Y 347.044,Z 383.389,A -85,B 0,C 180,E1 -13780.206,E2 -13780.206} C_VEL
LIN {X 0,Y 347.736,Z 376.693,A -85,B 0,C 180,E1 -13781.955,E2 -13781.955} C_VEL
LIN {X 0,Y 348.815,Z 368.395,A -85,B 0,C 180,E1 -13783.693,E2 -13783.693} C_VEL
LIN {X 0,Y 349.961,Z 359.091,A -85,B 0,C 180,E1 -13785.255,E2 -13785.255} C_VEL
LIN {X 0,Y 350.948,Z 349.376,A -85,B 0,C 180,E1 -13786.58,E2 -13786.58} C_VEL
LIN {X 0,Y 352.29,Z 337.554,A -85,B 0,C 180,E1 -13787.861,E2 -13787.861} C_VEL
LIN {X 0,Y 353.451,Z 325.658,A -85,B 0,C 180,E1 -13788.85,E2 -13788.85} C_VEL
LIN {X 0,Y 354.505,Z 313.283,A -85,B 0,C 180,E1 -13789.619,E2 -13789.619} C_VEL
LIN {X 0,Y 355.339,Z 300.56,A -85,B 0,C 180,E1 -13790.174,E2 -13790.174} C_VEL
LIN {X 0,Y 355.804,Z 287.169,A -85,B 0,C 180,E1 -13790.523,E2 -13790.523} C_VEL
LIN {X 0,Y 356.758,Z 222.967,A -85,B 0,C 180,E1 -13791.822,E2 -13791.822} C_VEL
LIN {X 0,Y 353.034,Z 198.658,A -85,B 0,C 180,E1 -13792.583,E2 -13792.583} C_VEL
LIN {X 0,Y 350.895,Z 186.556,A -85,B 0,C 180,E1 -13793.02,E2 -13793.02} C_VEL
LIN {X 0,Y 351.986,Z 176.311,A -85,B 0,C 180,E1 -13795.415,E2 -13795.415} C_VEL
LIN {X 0,Y 350.386,Z 167.062,A -85,B 0,C 180,E1 -13797.796,E2 -13797.796} C_VEL
LIN {X 0,Y 347.774,Z 155.166,A -85,B 0,C 180,E1 -13801.017,E2 -13801.017} C_VEL
LIN {X 0,Y 347.741,Z 155.166,A -85,B 0,C 180,E1 -13804.463,E2 -13804.463} C_VEL
LIN {X 0,Y 347.759,Z 155.164,A -85,B 0,C 180,E1 -13807.985,E2 -13807.985} C_VEL
LIN {X 0,Y 347.739,Z 155.167,A -85,B 0,C 180,E1 -13811.83,E2 -13811.83} C_VEL
LIN {X 0,Y 347.697,Z 155.175,A -85,B 0,C 180,E1 -13815.026,E2 -13815.026} C_VEL
LIN {X 0,Y 347.735,Z 155.167,A -85,B 0,C 180,E1 -13818.398,E2 -13818.398} C_VEL
LIN {X 0,Y 347.749,Z 155.167,A -85,B 0,C 180,E1 -13822.677,E2 -13822.677} C_VEL
LIN {X 0,Y 347.741,Z 155.165,A -85,B 0,C 180,E1 -13825.956,E2 -13825.956} C_VEL
LIN {X 0,Y 347.731,Z 155.167,A -85,B 0,C 180,E1 -13829.65,E2 -13829.65} C_VEL
LIN {X 0,Y 347.734,Z 155.166,A -85,B 0,C 180,E1 -13833.6,E2 -13833.6} C_VEL
LIN {X 0,Y 347.741,Z 155.167,A -85,B 0,C 180,E1 -13836.158,E2 -13836.158} C_VEL
LIN {X 0,Y 347.762,Z 155.164,A -85,B 0,C 180,E1 -13839.906,E2 -13839.906} C_VEL
LIN {X 0,Y 347.788,Z 155.158,A -85,B 0,C 180,E1 -13843.566,E2 -13843.566} C_VEL
LIN {X 0,Y 347.875,Z 155.149,A -85,B 0,C 180,E1 -13847.16,E2 -13847.16} C_VEL
LIN {X 0,Y 347.924,Z 155.144,A -85,B 0,C 180,E1 -13850.7,E2 -13850.7} C_VEL
LIN {X 0,Y 348.026,Z 155.135,A -85,B 0,C 180,E1 -13854.205,E2 -13854.205} C_VEL
LIN {X 0,Y 348.171,Z 155.113,A -85,B 0,C 180,E1 -13857.686,E2 -13857.686} C_VEL
LIN {X 0,Y 348.106,Z 155.121,A -85,B 0,C 180,E1 -13861.157,E2 -13861.157} C_VEL
LIN {X 0,Y 348.178,Z 155.113,A -85,B 0,C 180,E1 -13862.314,E2 -13862.314} C_VEL
LIN {X 0,Y 348.045,Z 155.127,A -85,B 0,C 180,E1 -13866.959,E2 -13866.959} C_VEL
LIN {X 0,Y 347.887,Z 155.147,A -85,B 0,C 180,E1 -13870.476,E2 -13870.476} C_VEL
LIN {X 0,Y 347.871,Z 155.15,A -85,B 0,C 180,E1 -13874.138,E2 -13874.138} C_VEL
LIN {X 0,Y 347.787,Z 155.159,A -85,B 0,C 180,E1 -13878.243,E2 -13878.243} C_VEL
LIN {X 0,Y 347.778,Z 155.164,A -85,B 0,C 180,E1 -13881.634,E2 -13881.634} C_VEL
LIN {X 0,Y 347.731,Z 155.171,A -85,B 0,C 180,E1 -13885.115,E2 -13885.115} C_VEL
LIN {X 0,Y 347.728,Z 155.169,A -85,B 0,C 180,E1 -13887.701,E2 -13887.701} C_VEL
LIN {X 0,Y 347.731,Z 155.167,A -85,B 0,C 180,E1 -13890.35,E2 -13890.35} C_VEL
LIN {X 0,Y 347.742,Z 155.166,A -85,B 0,C 180,E1 -13894.045,E2 -13894.045} C_VEL
LIN {X 0,Y 347.749,Z 155.167,A -85,B 0,C 180,E1 -13897.323,E2 -13897.323} C_VEL
LIN {X 0,Y 347.736,Z 155.167,A -85,B 0,C 180,E1 -13901.602,E2 -13901.602} C_VEL
LIN {X 0,Y 347.7,Z 155.173,A -85,B 0,C 180,E1 -13905.028,E2 -13905.028} C_VEL
LIN {X 0,Y 347.743,Z 155.169,A -85,B 0,C 180,E1 -13908.399,E2 -13908.399} C_VEL
LIN {X 0,Y 347.76,Z 155.164,A -85,B 0,C 180,E1 -13912.015,E2 -13912.015} C_VEL
LIN {X 0,Y 347.742,Z 155.166,A -85,B 0,C 180,E1 -13915.537,E2 -13915.537} C_VEL
LIN {X 0,Y 347.743,Z 155.171,A -85,B 0,C 180,E1 -13918.301,E2 -13918.301} C_VEL
LIN {X 0,Y 347.744,Z 155.165,A -85,B 0,C 180,E1 -13920.986,E2 -13920.986} C_VEL
LIN {X 0,Y 347.813,Z 155.276,A -85,B 0,C 180,E1 -13924.573,E2 -13924.573} C_VEL
LIN {X 0,Y 349.569,Z 163.53,A -85,B 0,C 180,E1 -13926.961,E2 -13926.961} C_VEL
LIN {X 0,Y 354.914,Z 177.663,A -85,B 0,C 180,E1 -13927.65,E2 -13927.65} C_VEL
LIN {X 0,Y 357.418,Z 190.394,A -85,B 0,C 180,E1 -13928.088,E2 -13928.088} C_VEL
LIN {X 0,Y 356.072,Z 265.871,A -85,B 0,C 180,E1 -13929.606,E2 -13929.606} C_VEL
LIN {X 0,Y 355.692,Z 278.747,A -85,B 0,C 180,E1 -13929.998,E2 -13929.998} C_VEL
LIN {X 0,Y 354.935,Z 291.98,A -85,B 0,C 180,E1 -13930.631,E2 -13930.631} C_VEL
LIN {X 0,Y 353.985,Z 304.357,A -85,B 0,C 180,E1 -13931.479,E2 -13931.479} C_VEL
LIN {X 0,Y 352.935,Z 315.447,A -85,B 0,C 180,E1 -13932.472,E2 -13932.472} C_VEL
LIN {X 0,Y 352.069,Z 325.128,A -85,B 0,C 180,E1 -13933.566,E2 -13933.566} C_VEL
LIN {X 0,Y 350.947,Z 334.896,A -85,B 0,C 180,E1 -13934.911,E2 -13934.911} C_VEL
LIN {X 0,Y 349.839,Z 343.382,A -85,B 0,C 180,E1 -13936.347,E2 -13936.347} C_VEL
LIN {X 0,Y 348.8,Z 351.623,A -85,B 0,C 180,E1 -13938.082,E2 -13938.082} C_VEL
LIN {X 0,Y 348.072,Z 357.26,A -85,B 0,C 180,E1 -13939.531,E2 -13939.531} C_VEL
LIN {X 0,Y 347.363,Z 362.753,A -85,B 0,C 180,E1 -13941.273,E2 -13941.273} C_VEL
LIN {X 0,Y 346.945,Z 367.06,A -85,B 0,C 180,E1 -13943.02,E2 -13943.02} C_VEL
LIN {X 0,Y 346.718,Z 369.339,A -85,B 0,C 180,E1 -13944.184,E2 -13944.184} C_VEL
LIN {X 0,Y 346.506,Z 371.195,A -85,B 0,C 180,E1 -13945.347,E2 -13945.347} C_VEL
LIN {X 0,Y 346.351,Z 372.591,A -85,B 0,C 180,E1 -13946.511,E2 -13946.511} C_VEL
LIN {X 0,Y 346.235,Z 374.193,A -85,B 0,C 180,E1 -13948.838,E2 -13948.838} C_VEL
LIN {X 0,Y 346.24,Z 374.425,A -85,B 0,C 180,E1 -13950.001,E2 -13950.001} C_VEL
LIN {X 0,Y 346.235,Z 374.236,A -85,B 0,C 180,E1 -13951.164,E2 -13951.164} C_VEL
LIN {X 0,Y 346.346,Z 372.688,A -85,B 0,C 180,E1 -13953.491,E2 -13953.491} C_VEL
LIN {X 0,Y 346.5,Z 371.334,A -85,B 0,C 180,E1 -13954.654,E2 -13954.654} C_VEL
LIN {X 0,Y 346.83,Z 368.322,A -85,B 0,C 180,E1 -13956.482,E2 -13956.482} C_VEL
LIN {X 0,Y 347.128,Z 364.597,A -85,B 0,C 180,E1 -13958.148,E2 -13958.148} C_VEL
LIN {X 0,Y 347.778,Z 359.588,A -85,B 0,C 180,E1 -13959.891,E2 -13959.891} C_VEL
LIN {X 0,Y 348.586,Z 353.282,A -85,B 0,C 180,E1 -13961.632,E2 -13961.632} C_VEL
LIN {X 0,Y 349.589,Z 345.386,A -85,B 0,C 180,E1 -13963.368,E2 -13963.368} C_VEL
LIN {X 0,Y 350.738,Z 337.329,A -85,B 0,C 180,E1 -13964.802,E2 -13964.802} C_VEL
LIN {X 0,Y 351.879,Z 327.502,A -85,B 0,C 180,E1 -13966.238,E2 -13966.238} C_VEL
LIN {X 0,Y 352.772,Z 317.834,A -85,B 0,C 180,E1 -13967.388,E2 -13967.388} C_VEL
LIN {X 0,Y 353.796,Z 307.358,A -85,B 0,C 180,E1 -13968.382,E2 -13968.382} C_VEL
LIN {X 0,Y 354.788,Z 294.739,A -85,B 0,C 180,E1 -13969.303,E2 -13969.303} C_VEL
LIN {X 0,Y 355.553,Z 282.1,A -85,B 0,C 180,E1 -13969.974,E2 -13969.974} C_VEL
LIN {X 0,Y 356.1,Z 270.081,A -85,B 0,C 180,E1 -13970.394,E2 -13970.394} C_VEL
LIN {X 0,Y 357.129,Z 212.448,A -85,B 0,C 180,E1 -13971.57,E2 -13971.57} C_VEL
LIN {X 0,Y 356.715,Z 206.597,A -85,B 0,C 180,E1 -13971.721,E2 -13971.721} C_VEL
LIN {X 0,Y 355.475,Z 200.901,A -85,B 0,C 180,E1 -13971.923,E2 -13971.923} C_VEL
LIN {X 0,Y 349.114,Z 182.489,A -85,B 0,C 180,E1 -13972.751,E2 -13972.751} C_VEL
LIN {X 0,Y 347.788,Z 177.643,A -85,B 0,C 180,E1 -13972.951,E2 -13972.951} C_VEL
LIN {X 0,Y 342.427,Z 163.839,A -85,B 0,C 180,E1 -13973.652,E2 -13973.652} C_VEL
LIN {X 0,Y 340.744,Z 156.042,A -85,B 0,C 180,E1 -13975.995,E2 -13975.995} C_VEL
LIN {X 0,Y 340.726,Z 156.044,A -85,B 0,C 180,E1 -13979.966,E2 -13979.966} C_VEL
LIN {X 0,Y 340.696,Z 156.047,A -85,B 0,C 180,E1 -13983.846,E2 -13983.846} C_VEL
LIN {X 0,Y 340.704,Z 156.042,A -85,B 0,C 180,E1 -13986.742,E2 -13986.742} C_VEL
LIN {X 0,Y 340.653,Z 156.05,A -85,B 0,C 180,E1 -13990.24,E2 -13990.24} C_VEL
LIN {X 0,Y 340.675,Z 156.048,A -85,B 0,C 180,E1 -13992.905,E2 -13992.905} C_VEL
LIN {X 0,Y 340.674,Z 156.049,A -85,B 0,C 180,E1 -13997.095,E2 -13997.095} C_VEL
LIN {X 0,Y 340.655,Z 156.047,A -85,B 0,C 180,E1 -14000.241,E2 -14000.241} C_VEL
LIN {X 0,Y 340.707,Z 156.043,A -85,B 0,C 180,E1 -14003.56,E2 -14003.56} C_VEL
LIN {X 0,Y 340.692,Z 156.043,A -85,B 0,C 180,E1 -14006.153,E2 -14006.153} C_VEL
LIN {X 0,Y 340.721,Z 156.039,A -85,B 0,C 180,E1 -14010.034,E2 -14010.034} C_VEL
LIN {X 0,Y 340.719,Z 156.045,A -85,B 0,C 180,E1 -14013.012,E2 -14013.012} C_VEL
LIN {X 0,Y 340.741,Z 156.037,A -85,B 0,C 180,E1 -14015.637,E2 -14015.637} C_VEL
LIN {X 0,Y 340.723,Z 156.04,A -85,B 0,C 180,E1 -14019.473,E2 -14019.473} C_VEL
LIN {X 0,Y 340.759,Z 156.036,A -85,B 0,C 180,E1 -14021.979,E2 -14021.979} C_VEL
LIN {X 0,Y 340.831,Z 156.024,A -85,B 0,C 180,E1 -14025.73,E2 -14025.73} C_VEL
LIN {X 0,Y 340.846,Z 156.025,A -85,B 0,C 180,E1 -14029.305,E2 -14029.305} C_VEL
LIN {X 0,Y 340.997,Z 156.003,A -85,B 0,C 180,E1 -14032.896,E2 -14032.896} C_VEL
LIN {X 0,Y 340.805,Z 156.029,A -85,B 0,C 180,E1 -14035.268,E2 -14035.268} C_VEL
LIN {X 0,Y 341.121,Z 155.992,A -85,B 0,C 180,E1 -14037.638,E2 -14037.638} C_VEL
LIN {X 0,Y 341.084,Z 155.992,A -85,B 0,C 180,E1 -14041.181,E2 -14041.181} C_VEL
LIN {X 0,Y 341.114,Z 155.993,A -85,B 0,C 180,E1 -14042.362,E2 -14042.362} C_VEL
LIN {X 0,Y 341.009,Z 156.01,A -85,B 0,C 180,E1 -14045.915,E2 -14045.915} C_VEL
LIN {X 0,Y 340.962,Z 156.009,A -85,B 0,C 180,E1 -14048.356,E2 -14048.356} C_VEL
LIN {X 0,Y 340.831,Z 156.031,A -85,B 0,C 180,E1 -14051.9,E2 -14051.9} C_VEL
LIN {X 0,Y 340.735,Z 156.043,A -85,B 0,C 180,E1 -14055.554,E2 -14055.554} C_VEL
LIN {X 0,Y 340.749,Z 156.036,A -85,B 0,C 180,E1 -14058.422,E2 -14058.422} C_VEL
LIN {X 0,Y 340.717,Z 156.042,A -85,B 0,C 180,E1 -14061.842,E2 -14061.842} C_VEL
LIN {X 0,Y 340.668,Z 156.05,A -85,B 0,C 180,E1 -14065.673,E2 -14065.673} C_VEL
LIN {X 0,Y 340.674,Z 156.045,A -85,B 0,C 180,E1 -14068.326,E2 -14068.326} C_VEL
LIN {X 0,Y 340.691,Z 156.048,A -85,B 0,C 180,E1 -14071.045,E2 -14071.045} C_VEL
LIN {X 0,Y 340.715,Z 156.045,A -85,B 0,C 180,E1 -14075.279,E2 -14075.279} C_VEL
LIN {X 0,Y 340.693,Z 156.043,A -85,B 0,C 180,E1 -14078.382,E2 -14078.382} C_VEL
LIN {X 0,Y 340.693,Z 156.043,A -85,B 0,C 180,E1 -14082.044,E2 -14082.044} C_VEL
LIN {X 0,Y 340.649,Z 156.051,A -85,B 0,C 180,E1 -14086.228,E2 -14086.228} C_VEL
LIN {X 0,Y 340.669,Z 156.052,A -85,B 0,C 180,E1 -14088.688,E2 -14088.688} C_VEL
LIN {X 0,Y 340.719,Z 156.04,A -85,B 0,C 180,E1 -14091.771,E2 -14091.771} C_VEL
LIN {X 0,Y 340.724,Z 156.041,A -85,B 0,C 180,E1 -14095.596,E2 -14095.596} C_VEL
LIN {X 0,Y 340.739,Z 156.09,A -85,B 0,C 180,E1 -14098.571,E2 -14098.571} C_VEL
LIN {X 0,Y 343.432,Z 168.174,A -85,B 0,C 180,E1 -14101.922,E2 -14101.922} C_VEL
LIN {X 0,Y 345.018,Z 176.923,A -85,B 0,C 180,E1 -14104.233,E2 -14104.233} C_VEL
LIN {X 0,Y 344.268,Z 185.295,A -85,B 0,C 180,E1 -14106.246,E2 -14106.246} C_VEL
LIN {X 0,Y 344.119,Z 186.427,A -85,B 0,C 180,E1 -14106.514,E2 -14106.514} C_VEL
LIN {X 0,Y 349.501,Z 218.312,A -85,B 0,C 180,E1 -14107.588,E2 -14107.588} C_VEL
LIN {X 0,Y 350.321,Z 224.749,A -85,B 0,C 180,E1 -14107.782,E2 -14107.782} C_VEL
LIN {X 0,Y 348.957,Z 295.178,A -85,B 0,C 180,E1 -14109.247,E2 -14109.247} C_VEL
LIN {X 0,Y 348.253,Z 308.376,A -85,B 0,C 180,E1 -14109.743,E2 -14109.743} C_VEL
LIN {X 0,Y 347.258,Z 320.5,A -85,B 0,C 180,E1 -14110.415,E2 -14110.415} C_VEL
LIN {X 0,Y 346.06,Z 332.741,A -85,B 0,C 180,E1 -14111.345,E2 -14111.345} C_VEL
LIN {X 0,Y 344.737,Z 344.33,A -85,B 0,C 180,E1 -14112.5,E2 -14112.5} C_VEL
LIN {X 0,Y 343.491,Z 354.773,A -85,B 0,C 180,E1 -14113.813,E2 -14113.813} C_VEL
LIN {X 0,Y 342.505,Z 363.312,A -85,B 0,C 180,E1 -14115.138,E2 -14115.138} C_VEL
LIN {X 0,Y 341.523,Z 371.195,A -85,B 0,C 180,E1 -14116.614,E2 -14116.614} C_VEL
LIN {X 0,Y 340.467,Z 378.893,A -85,B 0,C 180,E1 -14118.389,E2 -14118.389} C_VEL
LIN {X 0,Y 339.747,Z 386.004,A -85,B 0,C 180,E1 -14120.474,E2 -14120.474} C_VEL
LIN {X 0,Y 339.343,Z 390.736,A -85,B 0,C 180,E1 -14122.263,E2 -14122.263} C_VEL
LIN {X 0,Y 339.112,Z 394.529,A -85,B 0,C 180,E1 -14124.149,E2 -14124.149} C_VEL
LIN {X 0,Y 339.068,Z 396.222,A -85,B 0,C 180,E1 -14125.244,E2 -14125.244} C_VEL
LIN {X 0,Y 339.07,Z 397.624,A -85,B 0,C 180,E1 -14126.434,E2 -14126.434} C_VEL
LIN {X 0,Y 339.072,Z 399.234,A -85,B 0,C 180,E1 -14128.812,E2 -14128.812} C_VEL
LIN {X 0,Y 339.139,Z 399.452,A -85,B 0,C 180,E1 -14129.999,E2 -14129.999} C_VEL
LIN {X 0,Y 339.072,Z 399.229,A -85,B 0,C 180,E1 -14131.187,E2 -14131.187} C_VEL
LIN {X 0,Y 339.071,Z 397.613,A -85,B 0,C 180,E1 -14133.564,E2 -14133.564} C_VEL
LIN {X 0,Y 339.072,Z 396.206,A -85,B 0,C 180,E1 -14134.755,E2 -14134.755} C_VEL
LIN {X 0,Y 339.165,Z 393.253,A -85,B 0,C 180,E1 -14136.543,E2 -14136.543} C_VEL
LIN {X 0,Y 339.458,Z 389.261,A -85,B 0,C 180,E1 -14138.332,E2 -14138.332} C_VEL
LIN {X 0,Y 340.028,Z 383.127,A -85,B 0,C 180,E1 -14140.419,E2 -14140.419} C_VEL
LIN {X 0,Y 340.773,Z 376.431,A -85,B 0,C 180,E1 -14142.203,E2 -14142.203} C_VEL
LIN {X 0,Y 341.863,Z 368.132,A -85,B 0,C 180,E1 -14143.978,E2 -14143.978} C_VEL
LIN {X 0,Y 342.972,Z 359.625,A -85,B 0,C 180,E1 -14145.449,E2 -14145.449} C_VEL
LIN {X 0,Y 343.982,Z 350.29,A -85,B 0,C 180,E1 -14146.773,E2 -14146.773} C_VEL
LIN {X 0,Y 345.341,Z 338.72,A -85,B 0,C 180,E1 -14148.079,E2 -14148.079} C_VEL
LIN {X 0,Y 346.553,Z 327.328,A -85,B 0,C 180,E1 -14149.086,E2 -14149.086} C_VEL
LIN {X 0,Y 347.622,Z 315.62,A -85,B 0,C 180,E1 -14149.87,E2 -14149.87} C_VEL
LIN {X 0,Y 348.58,Z 302.126,A -85,B 0,C 180,E1 -14150.505,E2 -14150.505} C_VEL
LIN {X 0,Y 349.117,Z 288.68,A -85,B 0,C 180,E1 -14150.896,E2 -14150.896} C_VEL
LIN {X 0,Y 350.19,Z 223.839,A -85,B 0,C 180,E1 -14152.228,E2 -14152.228} C_VEL
LIN {X 0,Y 346.152,Z 197.843,A -85,B 0,C 180,E1 -14153.069,E2 -14153.069} C_VEL
LIN {X 0,Y 344.131,Z 186.319,A -85,B 0,C 180,E1 -14153.492,E2 -14153.492} C_VEL
LIN {X 0,Y 344.998,Z 178.624,A -85,B 0,C 180,E1 -14155.327,E2 -14155.327} C_VEL
LIN {X 0,Y 344.718,Z 175.078,A -85,B 0,C 180,E1 -14156.226,E2 -14156.226} C_VEL
LIN {X 0,Y 342.566,Z 164.112,A -85,B 0,C 180,E1 -14159.161,E2 -14159.161} C_VEL
LIN {X 0,Y 340.71,Z 156.047,A -85,B 0,C 180,E1 -14161.474,E2 -14161.474} C_VEL
LIN {X 0,Y 340.714,Z 156.044,A -85,B 0,C 180,E1 -14165.278,E2 -14165.278} C_VEL
LIN {X 0,Y 340.689,Z 156.043,A -85,B 0,C 180,E1 -14168.381,E2 -14168.381} C_VEL
LIN {X 0,Y 340.689,Z 156.044,A -85,B 0,C 180,E1 -14172.043,E2 -14172.043} C_VEL
LIN {X 0,Y 340.645,Z 156.05,A -85,B 0,C 180,E1 -14176.226,E2 -14176.226} C_VEL
LIN {X 0,Y 340.665,Z 156.049,A -85,B 0,C 180,E1 -14178.687,E2 -14178.687} C_VEL
LIN {X 0,Y 340.712,Z 156.042,A -85,B 0,C 180,E1 -14181.77,E2 -14181.77} C_VEL
LIN {X 0,Y 340.715,Z 156.041,A -85,B 0,C 180,E1 -14185.595,E2 -14185.595} C_VEL
LIN {X 0,Y 340.686,Z 156.049,A -85,B 0,C 180,E1 -14188.954,E2 -14188.954} C_VEL
LIN {X 0,Y 340.709,Z 156.044,A -85,B 0,C 180,E1 -14193.012,E2 -14193.012} C_VEL
LIN {X 0,Y 340.693,Z 156.045,A -85,B 0,C 180,E1 -14196.925,E2 -14196.925} C_VEL
LIN {X 0,Y 340.695,Z 156.047,A -85,B 0,C 180,E1 -14200.728,E2 -14200.728} C_VEL
LIN {X 0,Y 340.783,Z 156.037,A -85,B 0,C 180,E1 -14204.449,E2 -14204.449} C_VEL
LIN {X 0,Y 340.835,Z 156.03,A -85,B 0,C 180,E1 -14208.1,E2 -14208.1} C_VEL
LIN {X 0,Y 340.971,Z 156.009,A -85,B 0,C 180,E1 -14211.704,E2 -14211.704} C_VEL
LIN {X 0,Y 341.001,Z 156.011,A -85,B 0,C 180,E1 -14214.085,E2 -14214.085} C_VEL
LIN {X 0,Y 341.108,Z 155.992,A -85,B 0,C 180,E1 -14217.638,E2 -14217.638} C_VEL
LIN {X 0,Y 341.078,Z 155.996,A -85,B 0,C 180,E1 -14221.181,E2 -14221.181} C_VEL
LIN {X 0,Y 341.115,Z 155.992,A -85,B 0,C 180,E1 -14222.362,E2 -14222.362} C_VEL
LIN {X 0,Y 340.981,Z 156.008,A -85,B 0,C 180,E1 -14226.471,E2 -14226.471} C_VEL
LIN {X 0,Y 340.873,Z 156.025,A -85,B 0,C 180,E1 -14229.494,E2 -14229.494} C_VEL
LIN {X 0,Y 340.834,Z 156.025,A -85,B 0,C 180,E1 -14233.11,E2 -14233.11} C_VEL
LIN {X 0,Y 340.731,Z 156.039,A -85,B 0,C 180,E1 -14236.784,E2 -14236.784} C_VEL
LIN {X 0,Y 340.701,Z 156.046,A -85,B 0,C 180,E1 -14239.272,E2 -14239.272} C_VEL
LIN {X 0,Y 340.747,Z 156.039,A -85,B 0,C 180,E1 -14241.858,E2 -14241.858} C_VEL
LIN {X 0,Y 340.667,Z 156.047,A -85,B 0,C 180,E1 -14245.673,E2 -14245.673} C_VEL
LIN {X 0,Y 340.675,Z 156.046,A -85,B 0,C 180,E1 -14248.326,E2 -14248.326} C_VEL
LIN {X 0,Y 340.686,Z 156.049,A -85,B 0,C 180,E1 -14251.046,E2 -14251.046} C_VEL
LIN {X 0,Y 340.709,Z 156.045,A -85,B 0,C 180,E1 -14255.28,E2 -14255.28} C_VEL
LIN {X 0,Y 340.688,Z 156.046,A -85,B 0,C 180,E1 -14258.383,E2 -14258.383} C_VEL
LIN {X 0,Y 340.688,Z 156.045,A -85,B 0,C 180,E1 -14262.045,E2 -14262.045} C_VEL
LIN {X 0,Y 340.647,Z 156.051,A -85,B 0,C 180,E1 -14266.228,E2 -14266.228} C_VEL
LIN {X 0,Y 340.67,Z 156.047,A -85,B 0,C 180,E1 -14269.757,E2 -14269.757} C_VEL
LIN {X 0,Y 340.7,Z 156.044,A -85,B 0,C 180,E1 -14273.259,E2 -14273.259} C_VEL
LIN {X 0,Y 340.69,Z 156.048,A -85,B 0,C 180,E1 -14276.154,E2 -14276.154} C_VEL
LIN {X 0,Y 340.722,Z 156.043,A -85,B 0,C 180,E1 -14280.035,E2 -14280.035} C_VEL
LIN {X 0,Y 340.74,Z 156.119,A -85,B 0,C 180,E1 -14284.17,E2 -14284.17} C_VEL
LIN {X 0,Y 342.461,Z 164.017,A -85,B 0,C 180,E1 -14286.472,E2 -14286.472} C_VEL
LIN {X 0,Y 348.67,Z 180.331,A -85,B 0,C 180,E1 -14287.28,E2 -14287.28} C_VEL
LIN {X 0,Y 350.853,Z 191.57,A -85,B 0,C 180,E1 -14287.675,E2 -14287.675} C_VEL
LIN {X 0,Y 349.361,Z 269.155,A -85,B 0,C 180,E1 -14289.273,E2 -14289.273} C_VEL
LIN {X 0,Y 348.85,Z 282.499,A -85,B 0,C 180,E1 -14289.742,E2 -14289.742} C_VEL
LIN {X 0,Y 348.118,Z 294.534,A -85,B 0,C 180,E1 -14290.39,E2 -14290.39} C_VEL
LIN {X 0,Y 347.092,Z 306.384,A -85,B 0,C 180,E1 -14291.251,E2 -14291.251} C_VEL
LIN {X 0,Y 346.048,Z 317.13,A -85,B 0,C 180,E1 -14292.264,E2 -14292.264} C_VEL
LIN {X 0,Y 345.025,Z 328.073,A -85,B 0,C 180,E1 -14293.584,E2 -14293.584} C_VEL
LIN {X 0,Y 343.88,Z 336.965,A -85,B 0,C 180,E1 -14294.897,E2 -14294.897} C_VEL
LIN {X 0,Y 342.752,Z 345.121,A -85,B 0,C 180,E1 -14296.362,E2 -14296.362} C_VEL
LIN {X 0,Y 341.673,Z 353.108,A -85,B 0,C 180,E1 -14298.131,E2 -14298.131} C_VEL
LIN {X 0,Y 340.821,Z 359.517,A -85,B 0,C 180,E1 -14299.906,E2 -14299.906} C_VEL
LIN {X 0,Y 340.167,Z 364.599,A -85,B 0,C 180,E1 -14301.685,E2 -14301.685} C_VEL
LIN {X 0,Y 339.843,Z 367.685,A -85,B 0,C 180,E1 -14303.05,E2 -14303.05} C_VEL
LIN {X 0,Y 339.45,Z 371.454,A -85,B 0,C 180,E1 -14305.25,E2 -14305.25} C_VEL
LIN {X 0,Y 339.274,Z 372.851,A -85,B 0,C 180,E1 -14306.438,E2 -14306.438} C_VEL
LIN {X 0,Y 339.14,Z 374.453,A -85,B 0,C 180,E1 -14308.813,E2 -14308.813} C_VEL
LIN {X 0,Y 339.145,Z 374.684,A -85,B 0,C 180,E1 -14310.001,E2 -14310.001} C_VEL
LIN {X 0,Y 339.14,Z 374.494,A -85,B 0,C 180,E1 -14311.188,E2 -14311.188} C_VEL
LIN {X 0,Y 339.269,Z 372.946,A -85,B 0,C 180,E1 -14313.564,E2 -14313.564} C_VEL
LIN {X 0,Y 339.443,Z 371.592,A -85,B 0,C 180,E1 -14314.751,E2 -14314.751} C_VEL
LIN {X 0,Y 339.86,Z 367.857,A -85,B 0,C 180,E1 -14316.973,E2 -14316.973} C_VEL
LIN {X 0,Y 340.291,Z 363.3,A -85,B 0,C 180,E1 -14318.911,E2 -14318.911} C_VEL
LIN {X 0,Y 341.246,Z 356.869,A -85,B 0,C 180,E1 -14320.983,E2 -14320.983} C_VEL
LIN {X 0,Y 342.159,Z 349.805,A -85,B 0,C 180,E1 -14322.757,E2 -14322.757} C_VEL
LIN {X 0,Y 343.36,Z 340.998,A -85,B 0,C 180,E1 -14324.522,E2 -14324.522} C_VEL
LIN {X 0,Y 344.589,Z 331.956,A -85,B 0,C 180,E1 -14325.982,E2 -14325.982} C_VEL
LIN {X 0,Y 345.665,Z 321.713,A -85,B 0,C 180,E1 -14327.327,E2 -14327.327} C_VEL
LIN {X 0,Y 346.78,Z 310.805,A -85,B 0,C 180,E1 -14328.462,E2 -14328.462} C_VEL
LIN {X 0,Y 347.75,Z 300.274,A -85,B 0,C 180,E1 -14329.326,E2 -14329.326} C_VEL
LIN {X 0,Y 348.614,Z 287.587,A -85,B 0,C 180,E1 -14330.12,E2 -14330.12} C_VEL
LIN {X 0,Y 349.21,Z 276.058,A -85,B 0,C 180,E1 -14330.622,E2 -14330.622} C_VEL
LIN {X 0,Y 349.68,Z 261.475,A -85,B 0,C 180,E1 -14330.997,E2 -14330.997} C_VEL
LIN {X 0,Y 350.874,Z 190.965,A -85,B 0,C 180,E1 -14332.445,E2 -14332.445} C_VEL
LIN {X 0,Y 349.114,Z 182.489,A -85,B 0,C 180,E1 -14332.751,E2 -14332.751} C_VEL
LIN {X 0,Y 347.443,Z 179.115,A -85,B 0,C 180,E1 -14332.943,E2 -14332.943} C_VEL
LIN {X 0,Y 343.276,Z 174.524,A -85,B 0,C 180,E1 -14333.343,E2 -14333.343} C_VEL
LIN {X 0,Y 337.906,Z 169.213,A -85,B 0,C 180,E1 -14333.862,E2 -14333.862} C_VEL
LIN {X 0,Y 336.463,Z 167.124,A -85,B 0,C 180,E1 -14334.02,E2 -14334.02} C_VEL
LIN {X 0,Y 335.265,Z 164.056,A -85,B 0,C 180,E1 -14334.205,E2 -14334.205} C_VEL
LIN {X 0,Y 333.7,Z 156.919,A -85,B 0,C 180,E1 -14336.418,E2 -14336.418} C_VEL
LIN {X 0,Y 333.66,Z 156.922,A -85,B 0,C 180,E1 -14340.366,E2 -14340.366} C_VEL
LIN {X 0,Y 333.641,Z 156.924,A -85,B 0,C 180,E1 -14343.208,E2 -14343.208} C_VEL
LIN {X 0,Y 333.676,Z 156.919,A -85,B 0,C 180,E1 -14346.139,E2 -14346.139} C_VEL
LIN {X 0,Y 333.621,Z 156.928,A -85,B 0,C 180,E1 -14349.196,E2 -14349.196} C_VEL
LIN {X 0,Y 333.63,Z 156.924,A -85,B 0,C 180,E1 -14352.499,E2 -14352.499} C_VEL
LIN {X 0,Y 333.596,Z 156.928,A -85,B 0,C 180,E1 -14355.955,E2 -14355.955} C_VEL
LIN {X 0,Y 333.603,Z 156.93,A -85,B 0,C 180,E1 -14359.324,E2 -14359.324} C_VEL
LIN {X 0,Y 333.661,Z 156.924,A -85,B 0,C 180,E1 -14363.169,E2 -14363.169} C_VEL
LIN {X 0,Y 333.672,Z 156.92,A -85,B 0,C 180,E1 -14365.341,E2 -14365.341} C_VEL
LIN {X 0,Y 333.628,Z 156.924,A -85,B 0,C 180,E1 -14368.221,E2 -14368.221} C_VEL
LIN {X 0,Y 333.652,Z 156.923,A -85,B 0,C 180,E1 -14371.022,E2 -14371.022} C_VEL
LIN {X 0,Y 333.696,Z 156.917,A -85,B 0,C 180,E1 -14375.088,E2 -14375.088} C_VEL
LIN {X 0,Y 333.666,Z 156.921,A -85,B 0,C 180,E1 -14379.018,E2 -14379.018} C_VEL
LIN {X 0,Y 333.684,Z 156.918,A -85,B 0,C 180,E1 -14382.85,E2 -14382.85} C_VEL
LIN {X 0,Y 333.785,Z 156.908,A -85,B 0,C 180,E1 -14386.608,E2 -14386.608} C_VEL
LIN {X 0,Y 333.819,Z 156.905,A -85,B 0,C 180,E1 -14390.304,E2 -14390.304} C_VEL
LIN {X 0,Y 333.953,Z 156.881,A -85,B 0,C 180,E1 -14392.746,E2 -14392.746} C_VEL
LIN {X 0,Y 333.772,Z 156.905,A -85,B 0,C 180,E1 -14395.168,E2 -14395.168} C_VEL
LIN {X 0,Y 334.062,Z 156.871,A -85,B 0,C 180,E1 -14397.588,E2 -14397.588} C_VEL
LIN {X 0,Y 334.055,Z 156.866,A -85,B 0,C 180,E1 -14401.205,E2 -14401.205} C_VEL
LIN {X 0,Y 334.055,Z 156.871,A -85,B 0,C 180,E1 -14402.411,E2 -14402.411} C_VEL
LIN {X 0,Y 333.983,Z 156.883,A -85,B 0,C 180,E1 -14406.04,E2 -14406.04} C_VEL
LIN {X 0,Y 333.912,Z 156.886,A -85,B 0,C 180,E1 -14408.472,E2 -14408.472} C_VEL
LIN {X 0,Y 333.769,Z 156.908,A -85,B 0,C 180,E1 -14412.155,E2 -14412.155} C_VEL
LIN {X 0,Y 333.732,Z 156.91,A -85,B 0,C 180,E1 -14414.638,E2 -14414.638} C_VEL
LIN {X 0,Y 333.688,Z 156.916,A -85,B 0,C 180,E1 -14418.6,E2 -14418.6} C_VEL
LIN {X 0,Y 333.647,Z 156.92,A -85,B 0,C 180,E1 -14422.281,E2 -14422.281} C_VEL
LIN {X 0,Y 333.656,Z 156.922,A -85,B 0,C 180,E1 -14425.078,E2 -14425.078} C_VEL
LIN {X 0,Y 333.647,Z 156.923,A -85,B 0,C 180,E1 -14428.978,E2 -14428.978} C_VEL
LIN {X 0,Y 333.643,Z 156.923,A -85,B 0,C 180,E1 -14432.587,E2 -14432.587} C_VEL
LIN {X 0,Y 333.673,Z 156.919,A -85,B 0,C 180,E1 -14436.139,E2 -14436.139} C_VEL
LIN {X 0,Y 333.619,Z 156.929,A -85,B 0,C 180,E1 -14439.196,E2 -14439.196} C_VEL
LIN {X 0,Y 333.628,Z 156.926,A -85,B 0,C 180,E1 -14442.499,E2 -14442.499} C_VEL
LIN {X 0,Y 333.593,Z 156.929,A -85,B 0,C 180,E1 -14445.954,E2 -14445.954} C_VEL
LIN {X 0,Y 333.602,Z 156.927,A -85,B 0,C 180,E1 -14449.325,E2 -14449.325} C_VEL
LIN {X 0,Y 333.663,Z 156.921,A -85,B 0,C 180,E1 -14453.169,E2 -14453.169} C_VEL
LIN {X 0,Y 333.675,Z 156.92,A -85,B 0,C 180,E1 -14455.341,E2 -14455.341} C_VEL
LIN {X 0,Y 333.682,Z 157.025,A -85,B 0,C 180,E1 -14458.157,E2 -14458.157} C_VEL
LIN {X 0,Y 336.442,Z 169.114,A -85,B 0,C 180,E1 -14461.601,E2 -14461.601} C_VEL
LIN {X 0,Y 338.11,Z 178.431,A -85,B 0,C 180,E1 -14464.118,E2 -14464.118} C_VEL
LIN {X 0,Y 337.374,Z 186.135,A -85,B 0,C 180,E1 -14466.008,E2 -14466.008} C_VEL
LIN {X 0,Y 342.275,Z 215.146,A -85,B 0,C 180,E1 -14467.023,E2 -14467.023} C_VEL
LIN {X 0,Y 343.737,Z 225.634,A -85,B 0,C 180,E1 -14467.358,E2 -14467.358} C_VEL
LIN {X 0,Y 342.341,Z 294.932,A -85,B 0,C 180,E1 -14468.827,E2 -14468.827} C_VEL
LIN {X 0,Y 341.59,Z 308.125,A -85,B 0,C 180,E1 -14469.33,E2 -14469.33} C_VEL
LIN {X 0,Y 340.577,Z 320.247,A -85,B 0,C 180,E1 -14470.015,E2 -14470.015} C_VEL
LIN {X 0,Y 339.325,Z 332.486,A -85,B 0,C 180,E1 -14470.961,E2 -14470.961} C_VEL
LIN {X 0,Y 337.949,Z 344.073,A -85,B 0,C 180,E1 -14472.137,E2 -14472.137} C_VEL
LIN {X 0,Y 336.6,Z 354.834,A -85,B 0,C 180,E1 -14473.519,E2 -14473.519} C_VEL
LIN {X 0,Y 335.374,Z 364.753,A -85,B 0,C 180,E1 -14475.129,E2 -14475.129} C_VEL
LIN {X 0,Y 334.175,Z 373.676,A -85,B 0,C 180,E1 -14476.933,E2 -14476.933} C_VEL
LIN {X 0,Y 333.235,Z 380.878,A -85,B 0,C 180,E1 -14478.75,E2 -14478.75} C_VEL
LIN {X 0,Y 332.547,Z 387.444,A -85,B 0,C 180,E1 -14480.879,E2 -14480.879} C_VEL
LIN {X 0,Y 332.178,Z 391.791,A -85,B 0,C 180,E1 -14482.706,E2 -14482.706} C_VEL
LIN {X 0,Y 332.024,Z 394.55,A -85,B 0,C 180,E1 -14484.187,E2 -14484.187} C_VEL
LIN {X 0,Y 331.995,Z 397.366,A -85,B 0,C 180,E1 -14486.358,E2 -14486.358} C_VEL
LIN {X 0,Y 331.975,Z 398.975,A -85,B 0,C 180,E1 -14488.786,E2 -14488.786} C_VEL
LIN {X 0,Y 332.043,Z 399.192,A -85,B 0,C 180,E1 -14489.999,E2 -14489.999} C_VEL
LIN {X 0,Y 331.974,Z 398.97,A -85,B 0,C 180,E1 -14491.212,E2 -14491.212} C_VEL
LIN {X 0,Y 331.996,Z 397.354,A -85,B 0,C 180,E1 -14493.64,E2 -14493.64} C_VEL
LIN {X 0,Y 332.008,Z 394.57,A -85,B 0,C 180,E1 -14495.785,E2 -14495.785} C_VEL
LIN {X 0,Y 332.307,Z 390.439,A -85,B 0,C 180,E1 -14497.901,E2 -14497.901} C_VEL
LIN {X 0,Y 332.723,Z 385.695,A -85,B 0,C 180,E1 -14499.728,E2 -14499.728} C_VEL
LIN {X 0,Y 333.487,Z 378.575,A -85,B 0,C 180,E1 -14501.856,E2 -14501.856} C_VEL
LIN {X 0,Y 334.595,Z 370.857,A -85,B 0,C 180,E1 -14503.667,E2 -14503.667} C_VEL
LIN {X 0,Y 335.622,Z 362.964,A -85,B 0,C 180,E1 -14505.172,E2 -14505.172} C_VEL
LIN {X 0,Y 336.88,Z 352.351,A -85,B 0,C 180,E1 -14506.809,E2 -14506.809} C_VEL
LIN {X 0,Y 338.252,Z 341.312,A -85,B 0,C 180,E1 -14508.158,E2 -14508.158} C_VEL
LIN {X 0,Y 339.675,Z 328.835,A -85,B 0,C 180,E1 -14509.331,E2 -14509.331} C_VEL
LIN {X 0,Y 340.85,Z 316.583,A -85,B 0,C 180,E1 -14510.203,E2 -14510.203} C_VEL
LIN {X 0,Y 341.84,Z 303.688,A -85,B 0,C 180,E1 -14510.85,E2 -14510.85} C_VEL
LIN {X 0,Y 342.409,Z 289.965,A -85,B 0,C 180,E1 -14511.286,E2 -14511.286} C_VEL
LIN {X 0,Y 343.537,Z 224.096,A -85,B 0,C 180,E1 -14512.67,E2 -14512.67} C_VEL
LIN {X 0,Y 339.632,Z 199.018,A -85,B 0,C 180,E1 -14513.506,E2 -14513.506} C_VEL
LIN {X 0,Y 337.341,Z 186.132,A -85,B 0,C 180,E1 -14513.973,E2 -14513.973} C_VEL
LIN {X 0,Y 338.091,Z 178.348,A -85,B 0,C 180,E1 -14515.882,E2 -14515.882} C_VEL
LIN {X 0,Y 336.13,Z 167.798,A -85,B 0,C 180,E1 -14518.743,E2 -14518.743} C_VEL
LIN {X 0,Y 333.683,Z 156.921,A -85,B 0,C 180,E1 -14521.911,E2 -14521.911} C_VEL
LIN {X 0,Y 333.682,Z 156.917,A -85,B 0,C 180,E1 -14524.773,E2 -14524.773} C_VEL
LIN {X 0,Y 333.639,Z 156.924,A -85,B 0,C 180,E1 -14527.651,E2 -14527.651} C_VEL
LIN {X 0,Y 333.599,Z 156.928,A -85,B 0,C 180,E1 -14530.773,E2 -14530.773} C_VEL
LIN {X 0,Y 333.586,Z 156.929,A -85,B 0,C 180,E1 -14534.249,E2 -14534.249} C_VEL
LIN {X 0,Y 333.632,Z 156.926,A -85,B 0,C 180,E1 -14537.617,E2 -14537.617} C_VEL
LIN {X 0,Y 333.628,Z 156.928,A -85,B 0,C 180,E1 -14541.205,E2 -14541.205} C_VEL
LIN {X 0,Y 333.667,Z 156.919,A -85,B 0,C 180,E1 -14543.86,E2 -14543.86} C_VEL
LIN {X 0,Y 333.637,Z 156.923,A -85,B 0,C 180,E1 -14547.412,E2 -14547.412} C_VEL
LIN {X 0,Y 333.645,Z 156.922,A -85,B 0,C 180,E1 -14551.022,E2 -14551.022} C_VEL
LIN {X 0,Y 333.656,Z 156.922,A -85,B 0,C 180,E1 -14555.085,E2 -14555.085} C_VEL
LIN {X 0,Y 333.643,Z 156.924,A -85,B 0,C 180,E1 -14559.017,E2 -14559.017} C_VEL
LIN {X 0,Y 333.703,Z 156.914,A -85,B 0,C 180,E1 -14561.584,E2 -14561.584} C_VEL
LIN {X 0,Y 333.765,Z 156.907,A -85,B 0,C 180,E1 -14565.6,E2 -14565.6} C_VEL
LIN {X 0,Y 333.804,Z 156.9,A -85,B 0,C 180,E1 -14569.077,E2 -14569.077} C_VEL
LIN {X 0,Y 333.945,Z 156.885,A -85,B 0,C 180,E1 -14572.746,E2 -14572.746} C_VEL
LIN {X 0,Y 333.764,Z 156.906,A -85,B 0,C 180,E1 -14575.168,E2 -14575.168} C_VEL
LIN {X 0,Y 334.048,Z 156.87,A -85,B 0,C 180,E1 -14577.588,E2 -14577.588} C_VEL
LIN {X 0,Y 334.048,Z 156.872,A -85,B 0,C 180,E1 -14581.206,E2 -14581.206} C_VEL
LIN {X 0,Y 334.055,Z 156.871,A -85,B 0,C 180,E1 -14582.412,E2 -14582.412} C_VEL
LIN {X 0,Y 333.951,Z 156.883,A -85,B 0,C 180,E1 -14586.462,E2 -14586.462} C_VEL
LIN {X 0,Y 333.812,Z 156.906,A -85,B 0,C 180,E1 -14589.697,E2 -14589.697} C_VEL
LIN {X 0,Y 333.778,Z 156.905,A -85,B 0,C 180,E1 -14593.392,E2 -14593.392} C_VEL
LIN {X 0,Y 333.677,Z 156.92,A -85,B 0,C 180,E1 -14597.15,E2 -14597.15} C_VEL
LIN {X 0,Y 333.659,Z 156.92,A -85,B 0,C 180,E1 -14600.982,E2 -14600.982} C_VEL
LIN {X 0,Y 333.657,Z 156.922,A -85,B 0,C 180,E1 -14604.915,E2 -14604.915} C_VEL
LIN {X 0,Y 333.646,Z 156.926,A -85,B 0,C 180,E1 -14608.978,E2 -14608.978} C_VEL
LIN {X 0,Y 333.637,Z 156.923,A -85,B 0,C 180,E1 -14612.588,E2 -14612.588} C_VEL
LIN {X 0,Y 333.667,Z 156.919,A -85,B 0,C 180,E1 -14616.14,E2 -14616.14} C_VEL
LIN {X 0,Y 333.614,Z 156.928,A -85,B 0,C 180,E1 -14619.197,E2 -14619.197} C_VEL
LIN {X 0,Y 333.624,Z 156.927,A -85,B 0,C 180,E1 -14622.5,E2 -14622.5} C_VEL
LIN {X 0,Y 333.591,Z 156.928,A -85,B 0,C 180,E1 -14625.956,E2 -14625.956} C_VEL
LIN {X 0,Y 333.639,Z 156.923,A -85,B 0,C 180,E1 -14629.317,E2 -14629.317} C_VEL
LIN {X 0,Y 333.66,Z 156.921,A -85,B 0,C 180,E1 -14633.169,E2 -14633.169} C_VEL
LIN {X 0,Y 333.671,Z 156.919,A -85,B 0,C 180,E1 -14635.342,E2 -14635.342} C_VEL
LIN {X 0,Y 333.628,Z 156.929,A -85,B 0,C 180,E1 -14638.223,E2 -14638.223} C_VEL
LIN {X 0,Y 333.653,Z 156.92,A -85,B 0,C 180,E1 -14641.024,E2 -14641.024} C_VEL
LIN {X 0,Y 333.685,Z 156.969,A -85,B 0,C 180,E1 -14643.751,E2 -14643.751} C_VEL
LIN {X 0,Y 335.299,Z 164.141,A -85,B 0,C 180,E1 -14645.934,E2 -14645.934} C_VEL
LIN {X 0,Y 342.416,Z 182.803,A -85,B 0,C 180,E1 -14646.89,E2 -14646.89} C_VEL
LIN {X 0,Y 344.312,Z 192.289,A -85,B 0,C 180,E1 -14647.237,E2 -14647.237} C_VEL
LIN {X 0,Y 342.722,Z 270.879,A -85,B 0,C 180,E1 -14648.892,E2 -14648.892} C_VEL
LIN {X 0,Y 342.172,Z 284.287,A -85,B 0,C 180,E1 -14649.407,E2 -14649.407} C_VEL
LIN {X 0,Y 341.442,Z 294.8,A -85,B 0,C 180,E1 -14649.99,E2 -14649.99} C_VEL
LIN {X 0,Y 340.397,Z 306.649,A -85,B 0,C 180,E1 -14650.868,E2 -14650.868} C_VEL
LIN {X 0,Y 339.31,Z 317.394,A -85,B 0,C 180,E1 -14651.9,E2 -14651.9} C_VEL
LIN {X 0,Y 338.332,Z 327.264,A -85,B 0,C 180,E1 -14653.094,E2 -14653.094} C_VEL
LIN {X 0,Y 337.032,Z 337.227,A -85,B 0,C 180,E1 -14654.582,E2 -14654.582} C_VEL
LIN {X 0,Y 335.862,Z 345.383,A -85,B 0,C 180,E1 -14656.077,E2 -14656.077} C_VEL
LIN {X 0,Y 334.724,Z 353.37,A -85,B 0,C 180,E1 -14657.881,E2 -14657.881} C_VEL
LIN {X 0,Y 333.837,Z 359.777,A -85,B 0,C 180,E1 -14659.693,E2 -14659.693} C_VEL
LIN {X 0,Y 333.152,Z 364.859,A -85,B 0,C 180,E1 -14661.509,E2 -14661.509} C_VEL
LIN {X 0,Y 332.76,Z 368.256,A -85,B 0,C 180,E1 -14663.055,E2 -14663.055} C_VEL
LIN {X 0,Y 332.395,Z 371.713,A -85,B 0,C 180,E1 -14665.149,E2 -14665.149} C_VEL
LIN {X 0,Y 332.201,Z 373.11,A -85,B 0,C 180,E1 -14666.362,E2 -14666.362} C_VEL
LIN {X 0,Y 332.046,Z 374.712,A -85,B 0,C 180,E1 -14668.788,E2 -14668.788} C_VEL
LIN {X 0,Y 332.05,Z 374.943,A -85,B 0,C 180,E1 -14670.001,E2 -14670.001} C_VEL
LIN {X 0,Y 332.046,Z 374.753,A -85,B 0,C 180,E1 -14671.213,E2 -14671.213} C_VEL
LIN {X 0,Y 332.197,Z 373.205,A -85,B 0,C 180,E1 -14673.64,E2 -14673.64} C_VEL
LIN {X 0,Y 332.389,Z 371.849,A -85,B 0,C 180,E1 -14674.852,E2 -14674.852} C_VEL
LIN {X 0,Y 332.786,Z 368.398,A -85,B 0,C 180,E1 -14676.982,E2 -14676.982} C_VEL
LIN {X 0,Y 333.279,Z 363.558,A -85,B 0,C 180,E1 -14679.1,E2 -14679.1} C_VEL
LIN {X 0,Y 334.256,Z 357.127,A -85,B 0,C 180,E1 -14681.215,E2 -14681.215} C_VEL
LIN {X 0,Y 335.24,Z 350.062,A -85,B 0,C 180,E1 -14683.025,E2 -14683.025} C_VEL
LIN {X 0,Y 336.502,Z 341.254,A -85,B 0,C 180,E1 -14684.824,E2 -14684.824} C_VEL
LIN {X 0,Y 337.787,Z 332.211,A -85,B 0,C 180,E1 -14686.313,E2 -14686.313} C_VEL
LIN {X 0,Y 338.834,Z 322.581,A -85,B 0,C 180,E1 -14687.612,E2 -14687.612} C_VEL
LIN {X 0,Y 340.064,Z 311.058,A -85,B 0,C 180,E1 -14688.84,E2 -14688.84} C_VEL
LIN {X 0,Y 341.078,Z 300.525,A -85,B 0,C 180,E1 -14689.72,E2 -14689.72} C_VEL
LIN {X 0,Y 341.981,Z 287.836,A -85,B 0,C 180,E1 -14690.527,E2 -14690.527} C_VEL
LIN {X 0,Y 342.6,Z 276.302,A -85,B 0,C 180,E1 -14691.039,E2 -14691.039} C_VEL
LIN {X 0,Y 343.108,Z 262.6,A -85,B 0,C 180,E1 -14691.399,E2 -14691.399} C_VEL
LIN {X 0,Y 344.312,Z 192.043,A -85,B 0,C 180,E1 -14692.878,E2 -14692.878} C_VEL
LIN {X 0,Y 341.816,Z 180.803,A -85,B 0,C 180,E1 -14693.309,E2 -14693.309} C_VEL
LIN {X 0,Y 336.463,Z 167.124,A -85,B 0,C 180,E1 -14694.02,E2 -14694.02} C_VEL
LIN {X 0,Y 334.672,Z 165.089,A -85,B 0,C 180,E1 -14694.271,E2 -14694.271} C_VEL
LIN {X 0,Y 330.347,Z 162.41,A -85,B 0,C 180,E1 -14695.115,E2 -14695.115} C_VEL
LIN {X 0,Y 327.551,Z 160.148,A -85,B 0,C 180,E1 -14696.032,E2 -14696.032} C_VEL
LIN {X 0,Y 326.675,Z 157.795,A -85,B 0,C 180,E1 -14696.864,E2 -14696.864} C_VEL
LIN {X 0,Y 326.614,Z 157.799,A -85,B 0,C 180,E1 -14700.603,E2 -14700.603} C_VEL
LIN {X 0,Y 326.609,Z 157.801,A -85,B 0,C 180,E1 -14704.019,E2 -14704.019} C_VEL
LIN {X 0,Y 326.624,Z 157.799,A -85,B 0,C 180,E1 -14707.237,E2 -14707.237} C_VEL
LIN {X 0,Y 326.545,Z 157.809,A -85,B 0,C 180,E1 -14711.124,E2 -14711.124} C_VEL
LIN {X 0,Y 326.562,Z 157.809,A -85,B 0,C 180,E1 -14713.526,E2 -14713.526} C_VEL
LIN {X 0,Y 326.574,Z 157.805,A -85,B 0,C 180,E1 -14717.028,E2 -14717.028} C_VEL
LIN {X 0,Y 326.582,Z 157.805,A -85,B 0,C 180,E1 -14721.385,E2 -14721.385} C_VEL
LIN {X 0,Y 326.617,Z 157.799,A -85,B 0,C 180,E1 -14724.852,E2 -14724.852} C_VEL
LIN {X 0,Y 326.607,Z 157.8,A -85,B 0,C 180,E1 -14727.455,E2 -14727.455} C_VEL
LIN {X 0,Y 326.615,Z 157.797,A -85,B 0,C 180,E1 -14730.336,E2 -14730.336} C_VEL
LIN {X 0,Y 326.641,Z 157.799,A -85,B 0,C 180,E1 -14734.644,E2 -14734.644} C_VEL
LIN {X 0,Y 326.631,Z 157.796,A -85,B 0,C 180,E1 -14738.544,E2 -14738.544} C_VEL
LIN {X 0,Y 326.631,Z 157.8,A -85,B 0,C 180,E1 -14742.468,E2 -14742.468} C_VEL
LIN {X 0,Y 326.742,Z 157.782,A -85,B 0,C 180,E1 -14746.314,E2 -14746.314} C_VEL
LIN {X 0,Y 326.782,Z 157.78,A -85,B 0,C 180,E1 -14750.093,E2 -14750.093} C_VEL
LIN {X 0,Y 326.937,Z 157.754,A -85,B 0,C 180,E1 -14753.83,E2 -14753.83} C_VEL
LIN {X 0,Y 327.005,Z 157.75,A -85,B 0,C 180,E1 -14757.536,E2 -14757.536} C_VEL
LIN {X 0,Y 327.025,Z 157.741,A -85,B 0,C 180,E1 -14761.231,E2 -14761.231} C_VEL
LIN {X 0,Y 326.733,Z 157.784,A -85,B 0,C 180,E1 -14763.7,E2 -14763.7} C_VEL
LIN {X 0,Y 326.938,Z 157.76,A -85,B 0,C 180,E1 -14766.17,E2 -14766.17} C_VEL
LIN {X 0,Y 326.777,Z 157.778,A -85,B 0,C 180,E1 -14769.907,E2 -14769.907} C_VEL
LIN {X 0,Y 326.72,Z 157.789,A -85,B 0,C 180,E1 -14773.687,E2 -14773.687} C_VEL
LIN {X 0,Y 326.619,Z 157.797,A -85,B 0,C 180,E1 -14777.532,E2 -14777.532} C_VEL
LIN {X 0,Y 326.6,Z 157.803,A -85,B 0,C 180,E1 -14781.458,E2 -14781.458} C_VEL
LIN {X 0,Y 326.599,Z 157.804,A -85,B 0,C 180,E1 -14785.491,E2 -14785.491} C_VEL
LIN {X 0,Y 326.612,Z 157.799,A -85,B 0,C 180,E1 -14789.664,E2 -14789.664} C_VEL
LIN {X 0,Y 326.616,Z 157.801,A -85,B 0,C 180,E1 -14792.946,E2 -14792.946} C_VEL
LIN {X 0,Y 326.61,Z 157.8,A -85,B 0,C 180,E1 -14795.52,E2 -14795.52} C_VEL
LIN {X 0,Y 326.587,Z 157.805,A -85,B 0,C 180,E1 -14799.222,E2 -14799.222} C_VEL
LIN {X 0,Y 326.573,Z 157.808,A -85,B 0,C 180,E1 -14802.971,E2 -14802.971} C_VEL
LIN {X 0,Y 326.571,Z 157.805,A -85,B 0,C 180,E1 -14807.029,E2 -14807.029} C_VEL
LIN {X 0,Y 326.582,Z 157.802,A -85,B 0,C 180,E1 -14811.386,E2 -14811.386} C_VEL
LIN {X 0,Y 326.62,Z 157.801,A -85,B 0,C 180,E1 -14814.851,E2 -14814.851} C_VEL
LIN {X 0,Y 326.648,Z 157.984,A -85,B 0,C 180,E1 -14817.734,E2 -14817.734} C_VEL
LIN {X 0,Y 329.251,Z 169.357,A -85,B 0,C 180,E1 -14821.064,E2 -14821.064} C_VEL
LIN {X 0,Y 331.134,Z 179.461,A -85,B 0,C 180,E1 -14823.87,E2 -14823.87} C_VEL
LIN {X 0,Y 330.92,Z 183.37,A -85,B 0,C 180,E1 -14824.865,E2 -14824.865} C_VEL
LIN {X 0,Y 330.629,Z 186.119,A -85,B 0,C 180,E1 -14825.499,E2 -14825.499} C_VEL
LIN {X 0,Y 335.672,Z 215.526,A -85,B 0,C 180,E1 -14826.559,E2 -14826.559} C_VEL
LIN {X 0,Y 337.153,Z 226.896,A -85,B 0,C 180,E1 -14826.924,E2 -14826.924} C_VEL
LIN {X 0,Y 335.741,Z 294.686,A -85,B 0,C 180,E1 -14828.39,E2 -14828.39} C_VEL
LIN {X 0,Y 334.952,Z 307.875,A -85,B 0,C 180,E1 -14828.901,E2 -14828.901} C_VEL
LIN {X 0,Y 333.905,Z 319.994,A -85,B 0,C 180,E1 -14829.598,E2 -14829.598} C_VEL
LIN {X 0,Y 332.607,Z 332.231,A -85,B 0,C 180,E1 -14830.561,E2 -14830.561} C_VEL
LIN {X 0,Y 331.177,Z 343.817,A -85,B 0,C 180,E1 -14831.759,E2 -14831.759} C_VEL
LIN {X 0,Y 329.793,Z 354.258,A -85,B 0,C 180,E1 -14833.121,E2 -14833.121} C_VEL
LIN {X 0,Y 328.698,Z 363.218,A -85,B 0,C 180,E1 -14834.574,E2 -14834.574} C_VEL
LIN {X 0,Y 327.46,Z 372.057,A -85,B 0,C 180,E1 -14836.344,E2 -14836.344} C_VEL
LIN {X 0,Y 326.364,Z 379.499,A -85,B 0,C 180,E1 -14838.195,E2 -14838.195} C_VEL
LIN {X 0,Y 325.675,Z 385.485,A -85,B 0,C 180,E1 -14840.058,E2 -14840.058} C_VEL
LIN {X 0,Y 325.209,Z 390.217,A -85,B 0,C 180,E1 -14841.924,E2 -14841.924} C_VEL
LIN {X 0,Y 324.955,Z 393.836,A -85,B 0,C 180,E1 -14843.791,E2 -14843.791} C_VEL
LIN {X 0,Y 324.886,Z 395.704,A -85,B 0,C 180,E1 -14845.035,E2 -14845.035} C_VEL
LIN {X 0,Y 324.899,Z 397.106,A -85,B 0,C 180,E1 -14846.279,E2 -14846.279} C_VEL
LIN {X 0,Y 324.88,Z 398.716,A -85,B 0,C 180,E1 -14848.76,E2 -14848.76} C_VEL
LIN {X 0,Y 324.947,Z 398.933,A -85,B 0,C 180,E1 -14849.999,E2 -14849.999} C_VEL
LIN {X 0,Y 324.88,Z 398.71,A -85,B 0,C 180,E1 -14851.239,E2 -14851.239} C_VEL
LIN {X 0,Y 324.9,Z 397.094,A -85,B 0,C 180,E1 -14853.72,E2 -14853.72} C_VEL
LIN {X 0,Y 324.912,Z 394.577,A -85,B 0,C 180,E1 -14855.73,E2 -14855.73} C_VEL
LIN {X 0,Y 325.143,Z 391.499,A -85,B 0,C 180,E1 -14857.451,E2 -14857.451} C_VEL
LIN {X 0,Y 325.522,Z 387.138,A -85,B 0,C 180,E1 -14859.318,E2 -14859.318} C_VEL
LIN {X 0,Y 326.087,Z 381.587,A -85,B 0,C 180,E1 -14861.184,E2 -14861.184} C_VEL
LIN {X 0,Y 327.038,Z 374.668,A -85,B 0,C 180,E1 -14863.04,E2 -14863.04} C_VEL
LIN {X 0,Y 328,Z 367.605,A -85,B 0,C 180,E1 -14864.581,E2 -14864.581} C_VEL
LIN {X 0,Y 329.192,Z 359.097,A -85,B 0,C 180,E1 -14866.113,E2 -14866.113} C_VEL
LIN {X 0,Y 330.539,Z 348.586,A -85,B 0,C 180,E1 -14867.636,E2 -14867.636} C_VEL
LIN {X 0,Y 331.875,Z 338.194,A -85,B 0,C 180,E1 -14868.84,E2 -14868.84} C_VEL
LIN {X 0,Y 333.156,Z 326.798,A -85,B 0,C 180,E1 -14869.886,E2 -14869.886} C_VEL
LIN {X 0,Y 334.303,Z 315.087,A -85,B 0,C 180,E1 -14870.697,E2 -14870.697} C_VEL
LIN {X 0,Y 335.34,Z 301.588,A -85,B 0,C 180,E1 -14871.354,E2 -14871.354} C_VEL
LIN {X 0,Y 335.886,Z 288.119,A -85,B 0,C 180,E1 -14871.76,E2 -14871.76} C_VEL
LIN {X 0,Y 336.988,Z 225.01,A -85,B 0,C 180,E1 -14873.109,E2 -14873.109} C_VEL
LIN {X 0,Y 333.119,Z 200.015,A -85,B 0,C 180,E1 -14873.964,E2 -14873.964} C_VEL
LIN {X 0,Y 330.551,Z 185.788,A -85,B 0,C 180,E1 -14874.516,E2 -14874.516} C_VEL
LIN {X 0,Y 331.206,Z 180.687,A -85,B 0,C 180,E1 -14875.784,E2 -14875.784} C_VEL
LIN {X 0,Y 329.633,Z 171.042,A -85,B 0,C 180,E1 -14878.431,E2 -14878.431} C_VEL
LIN {X 0,Y 326.643,Z 157.797,A -85,B 0,C 180,E1 -14882.311,E2 -14882.311} C_VEL
LIN {X 0,Y 326.609,Z 157.801,A -85,B 0,C 180,E1 -14885.519,E2 -14885.519} C_VEL
LIN {X 0,Y 326.584,Z 157.804,A -85,B 0,C 180,E1 -14889.221,E2 -14889.221} C_VEL
LIN {X 0,Y 326.568,Z 157.806,A -85,B 0,C 180,E1 -14892.97,E2 -14892.97} C_VEL
LIN {X 0,Y 326.567,Z 157.807,A -85,B 0,C 180,E1 -14897.028,E2 -14897.028} C_VEL
LIN {X 0,Y 326.576,Z 157.805,A -85,B 0,C 180,E1 -14901.385,E2 -14901.385} C_VEL
LIN {X 0,Y 326.611,Z 157.802,A -85,B 0,C 180,E1 -14904.851,E2 -14904.851} C_VEL
LIN {X 0,Y 326.601,Z 157.799,A -85,B 0,C 180,E1 -14907.455,E2 -14907.455} C_VEL
LIN {X 0,Y 326.608,Z 157.8,A -85,B 0,C 180,E1 -14910.336,E2 -14910.336} C_VEL
LIN {X 0,Y 326.594,Z 157.804,A -85,B 0,C 180,E1 -14914.508,E2 -14914.508} C_VEL
LIN {X 0,Y 326.6,Z 157.802,A -85,B 0,C 180,E1 -14918.542,E2 -14918.542} C_VEL
LIN {X 0,Y 326.623,Z 157.798,A -85,B 0,C 180,E1 -14922.468,E2 -14922.468} C_VEL
LIN {X 0,Y 326.733,Z 157.788,A -85,B 0,C 180,E1 -14926.314,E2 -14926.314} C_VEL
LIN {X 0,Y 326.772,Z 157.779,A -85,B 0,C 180,E1 -14930.092,E2 -14930.092} C_VEL
LIN {X 0,Y 326.93,Z 157.761,A -85,B 0,C 180,E1 -14933.83,E2 -14933.83} C_VEL
LIN {X 0,Y 326.991,Z 157.748,A -85,B 0,C 180,E1 -14937.536,E2 -14937.536} C_VEL
LIN {X 0,Y 327.019,Z 157.748,A -85,B 0,C 180,E1 -14941.232,E2 -14941.232} C_VEL
LIN {X 0,Y 326.741,Z 157.785,A -85,B 0,C 180,E1 -14943.7,E2 -14943.7} C_VEL
LIN {X 0,Y 326.913,Z 157.76,A -85,B 0,C 180,E1 -14946.45,E2 -14946.45} C_VEL
LIN {X 0,Y 326.775,Z 157.78,A -85,B 0,C 180,E1 -14949.908,E2 -14949.908} C_VEL
LIN {X 0,Y 326.734,Z 157.785,A -85,B 0,C 180,E1 -14953.687,E2 -14953.687} C_VEL
LIN {X 0,Y 326.624,Z 157.8,A -85,B 0,C 180,E1 -14957.532,E2 -14957.532} C_VEL
LIN {X 0,Y 326.624,Z 157.801,A -85,B 0,C 180,E1 -14961.456,E2 -14961.456} C_VEL
LIN {X 0,Y 326.594,Z 157.8,A -85,B 0,C 180,E1 -14965.492,E2 -14965.492} C_VEL
LIN {X 0,Y 326.609,Z 157.799,A -85,B 0,C 180,E1 -14969.664,E2 -14969.664} C_VEL
LIN {X 0,Y 326.611,Z 157.801,A -85,B 0,C 180,E1 -14972.947,E2 -14972.947} C_VEL
LIN {X 0,Y 326.604,Z 157.8,A -85,B 0,C 180,E1 -14975.521,E2 -14975.521} C_VEL
LIN {X 0,Y 326.582,Z 157.804,A -85,B 0,C 180,E1 -14979.223,E2 -14979.223} C_VEL
LIN {X 0,Y 326.569,Z 157.807,A -85,B 0,C 180,E1 -14982.972,E2 -14982.972} C_VEL
LIN {X 0,Y 326.571,Z 157.805,A -85,B 0,C 180,E1 -14987.029,E2 -14987.029} C_VEL
LIN {X 0,Y 326.595,Z 157.803,A -85,B 0,C 180,E1 -14990.777,E2 -14990.777} C_VEL
LIN {X 0,Y 326.61,Z 157.802,A -85,B 0,C 180,E1 -14994.481,E2 -14994.481} C_VEL
LIN {X 0,Y 326.606,Z 157.8,A -85,B 0,C 180,E1 -14997.457,E2 -14997.457} C_VEL
LIN {X 0,Y 326.615,Z 157.801,A -85,B 0,C 180,E1 -15000.338,E2 -15000.338} C_VEL
LIN {X 0,Y 326.638,Z 157.822,A -85,B 0,C 180,E1 -15003.312,E2 -15003.312} C_VEL
LIN {X 0,Y 328.111,Z 164.355,A -85,B 0,C 180,E1 -15005.355,E2 -15005.355} C_VEL
LIN {X 0,Y 336.106,Z 184.913,A -85,B 0,C 180,E1 -15006.472,E2 -15006.472} C_VEL
LIN {X 0,Y 337.787,Z 193.405,A -85,B 0,C 180,E1 -15006.791,E2 -15006.791} C_VEL
LIN {X 0,Y 336.148,Z 269.714,A -85,B 0,C 180,E1 -15008.419,E2 -15008.419} C_VEL
LIN {X 0,Y 335.588,Z 283.038,A -85,B 0,C 180,E1 -15008.904,E2 -15008.904} C_VEL
LIN {X 0,Y 334.796,Z 295.067,A -85,B 0,C 180,E1 -15009.575,E2 -15009.575} C_VEL
LIN {X 0,Y 333.712,Z 306.913,A -85,B 0,C 180,E1 -15010.469,E2 -15010.469} C_VEL
LIN {X 0,Y 332.57,Z 317.658,A -85,B 0,C 180,E1 -15011.52,E2 -15011.52} C_VEL
LIN {X 0,Y 331.542,Z 327.527,A -85,B 0,C 180,E1 -15012.737,E2 -15012.737} C_VEL
LIN {X 0,Y 330.191,Z 337.489,A -85,B 0,C 180,E1 -15014.255,E2 -15014.255} C_VEL
LIN {X 0,Y 328.797,Z 347.12,A -85,B 0,C 180,E1 -15016.087,E2 -15016.087} C_VEL
LIN {X 0,Y 327.634,Z 354.799,A -85,B 0,C 180,E1 -15017.929,E2 -15017.929} C_VEL
LIN {X 0,Y 326.869,Z 360.038,A -85,B 0,C 180,E1 -15019.47,E2 -15019.47} C_VEL
LIN {X 0,Y 326.124,Z 365.12,A -85,B 0,C 180,E1 -15021.325,E2 -15021.325} C_VEL
LIN {X 0,Y 325.664,Z 368.86,A -85,B 0,C 180,E1 -15023.077,E2 -15023.077} C_VEL
LIN {X 0,Y 325.342,Z 371.973,A -85,B 0,C 180,E1 -15025.044,E2 -15025.044} C_VEL
LIN {X 0,Y 325.132,Z 373.369,A -85,B 0,C 180,E1 -15026.283,E2 -15026.283} C_VEL
LIN {X 0,Y 324.952,Z 374.971,A -85,B 0,C 180,E1 -15028.761,E2 -15028.761} C_VEL
LIN {X 0,Y 324.955,Z 375.202,A -85,B 0,C 180,E1 -15030.001,E2 -15030.001} C_VEL
LIN {X 0,Y 324.951,Z 375.012,A -85,B 0,C 180,E1 -15031.24,E2 -15031.24} C_VEL
LIN {X 0,Y 325.127,Z 373.463,A -85,B 0,C 180,E1 -15033.719,E2 -15033.719} C_VEL
LIN {X 0,Y 325.337,Z 372.107,A -85,B 0,C 180,E1 -15034.958,E2 -15034.958} C_VEL
LIN {X 0,Y 325.705,Z 368.953,A -85,B 0,C 180,E1 -15036.983,E2 -15036.983} C_VEL
LIN {X 0,Y 326.258,Z 363.816,A -85,B 0,C 180,E1 -15039.298,E2 -15039.298} C_VEL
LIN {X 0,Y 327.268,Z 357.386,A -85,B 0,C 180,E1 -15041.458,E2 -15041.458} C_VEL
LIN {X 0,Y 328.298,Z 350.32,A -85,B 0,C 180,E1 -15043.305,E2 -15043.305} C_VEL
LIN {X 0,Y 329.655,Z 341.51,A -85,B 0,C 180,E1 -15045.139,E2 -15045.139} C_VEL
LIN {X 0,Y 330.988,Z 332.497,A -85,B 0,C 180,E1 -15046.653,E2 -15046.653} C_VEL
LIN {X 0,Y 332.128,Z 322.46,A -85,B 0,C 180,E1 -15048.027,E2 -15048.027} C_VEL
LIN {X 0,Y 333.37,Z 311.311,A -85,B 0,C 180,E1 -15049.233,E2 -15049.233} C_VEL
LIN {X 0,Y 334.429,Z 300.777,A -85,B 0,C 180,E1 -15050.128,E2 -15050.128} C_VEL
LIN {X 0,Y 335.358,Z 288.086,A -85,B 0,C 180,E1 -15050.952,E2 -15050.952} C_VEL
LIN {X 0,Y 336.011,Z 276.545,A -85,B 0,C 180,E1 -15051.471,E2 -15051.471} C_VEL
LIN {X 0,Y 336.499,Z 261.049,A -85,B 0,C 180,E1 -15051.881,E2 -15051.881} C_VEL
LIN {X 0,Y 337.787,Z 193.169,A -85,B 0,C 180,E1 -15053.326,E2 -15053.326} C_VEL
LIN {X 0,Y 335.6,Z 183.312,A -85,B 0,C 180,E1 -15053.715,E2 -15053.715} C_VEL
LIN {X 0,Y 328.103,Z 164.279,A -85,B 0,C 180,E1 -15054.783,E2 -15054.783} C_VEL
LIN {X 0,Y 326.675,Z 157.795,A -85,B 0,C 180,E1 -15056.864,E2 -15056.864} C_VEL
LIN {X 0,Y 325.934,Z 157.887,A -85,B 0,C 180,E1 -15057.893,E2 -15057.893} C_VEL
LIN {X 0,Y 323.031,Z 158.248,A -85,B 0,C 180,E1 -15059.568,E2 -15059.568} C_VEL
LIN {X 0,Y 320.618,Z 158.547,A -85,B 0,C 180,E1 -15060.925,E2 -15060.925} C_VEL
LIN {X 0,Y 319.599,Z 158.673,A -85,B 0,C 180,E1 -15061.975,E2 -15061.975} C_VEL
LIN {X 0,Y 319.522,Z 158.68,A -85,B 0,C 180,E1 -15062.331,E2 -15062.331} C_VEL
LIN {X 0,Y 319.581,Z 158.679,A -85,B 0,C 180,E1 -15065.543,E2 -15065.543} C_VEL
LIN {X 0,Y 319.529,Z 158.685,A -85,B 0,C 180,E1 -15069.662,E2 -15069.662} C_VEL
LIN {X 0,Y 319.521,Z 158.687,A -85,B 0,C 180,E1 -15073.46,E2 -15073.46} C_VEL
LIN {X 0,Y 319.553,Z 158.679,A -85,B 0,C 180,E1 -15077.016,E2 -15077.016} C_VEL
LIN {X 0,Y 319.545,Z 158.675,A -85,B 0,C 180,E1 -15080.37,E2 -15080.37} C_VEL
LIN {X 0,Y 319.578,Z 158.673,A -85,B 0,C 180,E1 -15084.458,E2 -15084.458} C_VEL
LIN {X 0,Y 319.524,Z 158.681,A -85,B 0,C 180,E1 -15088.137,E2 -15088.137} C_VEL
LIN {X 0,Y 319.57,Z 158.674,A -85,B 0,C 180,E1 -15091.604,E2 -15091.604} C_VEL
LIN {X 0,Y 319.574,Z 158.675,A -85,B 0,C 180,E1 -15095.301,E2 -15095.301} C_VEL
LIN {X 0,Y 319.588,Z 158.669,A -85,B 0,C 180,E1 -15098.047,E2 -15098.047} C_VEL
LIN {X 0,Y 319.586,Z 158.675,A -85,B 0,C 180,E1 -15102.069,E2 -15102.069} C_VEL
LIN {X 0,Y 319.708,Z 158.655,A -85,B 0,C 180,E1 -15106.007,E2 -15106.007} C_VEL
LIN {X 0,Y 319.734,Z 158.656,A -85,B 0,C 180,E1 -15109.872,E2 -15109.872} C_VEL
LIN {X 0,Y 319.895,Z 158.63,A -85,B 0,C 180,E1 -15113.693,E2 -15113.693} C_VEL
LIN {X 0,Y 319.952,Z 158.628,A -85,B 0,C 180,E1 -15117.482,E2 -15117.482} C_VEL
LIN {X 0,Y 319.994,Z 158.616,A -85,B 0,C 180,E1 -15121.258,E2 -15121.258} C_VEL
LIN {X 0,Y 319.71,Z 158.658,A -85,B 0,C 180,E1 -15125.044,E2 -15125.044} C_VEL
LIN {X 0,Y 319.851,Z 158.642,A -85,B 0,C 180,E1 -15127.576,E2 -15127.576} C_VEL
LIN {X 0,Y 319.701,Z 158.659,A -85,B 0,C 180,E1 -15131.411,E2 -15131.411} C_VEL
LIN {X 0,Y 319.648,Z 158.664,A -85,B 0,C 180,E1 -15134.668,E2 -15134.668} C_VEL
LIN {X 0,Y 319.597,Z 158.672,A -85,B 0,C 180,E1 -15138.99,E2 -15138.99} C_VEL
LIN {X 0,Y 319.579,Z 158.672,A -85,B 0,C 180,E1 -15142.536,E2 -15142.536} C_VEL
LIN {X 0,Y 319.548,Z 158.679,A -85,B 0,C 180,E1 -15146.096,E2 -15146.096} C_VEL
LIN {X 0,Y 319.539,Z 158.68,A -85,B 0,C 180,E1 -15148.939,E2 -15148.939} C_VEL
LIN {X 0,Y 319.523,Z 158.682,A -85,B 0,C 180,E1 -15151.863,E2 -15151.863} C_VEL
LIN {X 0,Y 319.578,Z 158.676,A -85,B 0,C 180,E1 -15155.542,E2 -15155.542} C_VEL
LIN {X 0,Y 319.528,Z 158.681,A -85,B 0,C 180,E1 -15159.662,E2 -15159.662} C_VEL
LIN {X 0,Y 319.519,Z 158.683,A -85,B 0,C 180,E1 -15163.46,E2 -15163.46} C_VEL
LIN {X 0,Y 319.55,Z 158.68,A -85,B 0,C 180,E1 -15167.016,E2 -15167.016} C_VEL
LIN {X 0,Y 319.545,Z 158.68,A -85,B 0,C 180,E1 -15170.371,E2 -15170.371} C_VEL
LIN {X 0,Y 319.58,Z 158.68,A -85,B 0,C 180,E1 -15174.457,E2 -15174.457} C_VEL
LIN {X 0,Y 319.589,Z 158.716,A -85,B 0,C 180,E1 -15177.222,E2 -15177.222} C_VEL
LIN {X 0,Y 322.24,Z 170.41,A -85,B 0,C 180,E1 -15180.738,E2 -15180.738} C_VEL
LIN {X 0,Y 324.155,Z 180.491,A -85,B 0,C 180,E1 -15183.611,E2 -15183.611} C_VEL
LIN {X 0,Y 324.06,Z 184.271,A -85,B 0,C 180,E1 -15184.604,E2 -15184.604} C_VEL
LIN {X 0,Y 323.864,Z 185.583,A -85,B 0,C 180,E1 -15184.936,E2 -15184.936} C_VEL
LIN {X 0,Y 328.892,Z 214.656,A -85,B 0,C 180,E1 -15186.031,E2 -15186.031} C_VEL
LIN {X 0,Y 330.614,Z 226.618,A -85,B 0,C 180,E1 -15186.44,E2 -15186.44} C_VEL
LIN {X 0,Y 329.137,Z 294.44,A -85,B 0,C 180,E1 -15187.934,E2 -15187.934} C_VEL
LIN {X 0,Y 328.345,Z 307.625,A -85,B 0,C 180,E1 -15188.456,E2 -15188.456} C_VEL
LIN {X 0,Y 327.252,Z 319.741,A -85,B 0,C 180,E1 -15189.164,E2 -15189.164} C_VEL
LIN {X 0,Y 325.902,Z 331.976,A -85,B 0,C 180,E1 -15190.144,E2 -15190.144} C_VEL
LIN {X 0,Y 324.432,Z 343.561,A -85,B 0,C 180,E1 -15191.366,E2 -15191.366} C_VEL
LIN {X 0,Y 322.972,Z 353.997,A -85,B 0,C 180,E1 -15192.753,E2 -15192.753} C_VEL
LIN {X 0,Y 321.77,Z 363.364,A -85,B 0,C 180,E1 -15194.311,E2 -15194.311} C_VEL
LIN {X 0,Y 320.522,Z 371.798,A -85,B 0,C 180,E1 -15196.043,E2 -15196.043} C_VEL
LIN {X 0,Y 319.386,Z 379.241,A -85,B 0,C 180,E1 -15197.933,E2 -15197.933} C_VEL
LIN {X 0,Y 318.638,Z 385.225,A -85,B 0,C 180,E1 -15199.836,E2 -15199.836} C_VEL
LIN {X 0,Y 318.167,Z 389.958,A -85,B 0,C 180,E1 -15201.744,E2 -15201.744} C_VEL
LIN {X 0,Y 317.882,Z 393.577,A -85,B 0,C 180,E1 -15203.653,E2 -15203.653} C_VEL
LIN {X 0,Y 317.801,Z 395.445,A -85,B 0,C 180,E1 -15204.925,E2 -15204.925} C_VEL
LIN {X 0,Y 317.806,Z 396.847,A -85,B 0,C 180,E1 -15206.195,E2 -15206.195} C_VEL
LIN {X 0,Y 317.779,Z 397.847,A -85,B 0,C 180,E1 -15207.464,E2 -15207.464} C_VEL
LIN {X 0,Y 317.788,Z 398.458,A -85,B 0,C 180,E1 -15208.732,E2 -15208.732} C_VEL
LIN {X 0,Y 317.851,Z 398.674,A -85,B 0,C 180,E1 -15209.999,E2 -15209.999} C_VEL
LIN {X 0,Y 317.788,Z 398.451,A -85,B 0,C 180,E1 -15211.267,E2 -15211.267} C_VEL
LIN {X 0,Y 317.779,Z 397.837,A -85,B 0,C 180,E1 -15212.534,E2 -15212.534} C_VEL
LIN {X 0,Y 317.807,Z 396.834,A -85,B 0,C 180,E1 -15213.803,E2 -15213.803} C_VEL
LIN {X 0,Y 317.837,Z 394.53,A -85,B 0,C 180,E1 -15215.708,E2 -15215.708} C_VEL
LIN {X 0,Y 318.062,Z 391.237,A -85,B 0,C 180,E1 -15217.618,E2 -15217.618} C_VEL
LIN {X 0,Y 318.465,Z 386.876,A -85,B 0,C 180,E1 -15219.526,E2 -15219.526} C_VEL
LIN {X 0,Y 319.076,Z 381.324,A -85,B 0,C 180,E1 -15221.433,E2 -15221.433} C_VEL
LIN {X 0,Y 320.095,Z 374.406,A -85,B 0,C 180,E1 -15223.328,E2 -15223.328} C_VEL
LIN {X 0,Y 321.376,Z 365.751,A -85,B 0,C 180,E1 -15225.213,E2 -15225.213} C_VEL
LIN {X 0,Y 322.565,Z 356.877,A -85,B 0,C 180,E1 -15226.779,E2 -15226.779} C_VEL
LIN {X 0,Y 323.884,Z 347.144,A -85,B 0,C 180,E1 -15228.174,E2 -15228.174} C_VEL
LIN {X 0,Y 325.362,Z 336.5,A -85,B 0,C 180,E1 -15229.396,E2 -15229.396} C_VEL
LIN {X 0,Y 326.667,Z 324.597,A -85,B 0,C 180,E1 -15230.462,E2 -15230.462} C_VEL
LIN {X 0,Y 327.881,Z 312.215,A -85,B 0,C 180,E1 -15231.287,E2 -15231.287} C_VEL
LIN {X 0,Y 328.858,Z 299.48,A -85,B 0,C 180,E1 -15231.878,E2 -15231.878} C_VEL
LIN {X 0,Y 329.366,Z 286.05,A -85,B 0,C 180,E1 -15232.255,E2 -15232.255} C_VEL
LIN {X 0,Y 330.454,Z 225.838,A -85,B 0,C 180,E1 -15233.567,E2 -15233.567} C_VEL
LIN {X 0,Y 326.484,Z 200.232,A -85,B 0,C 180,E1 -15234.471,E2 -15234.471} C_VEL
LIN {X 0,Y 323.819,Z 185.5,A -85,B 0,C 180,E1 -15235.065,E2 -15235.065} C_VEL
LIN {X 0,Y 324.291,Z 181.715,A -85,B 0,C 180,E1 -15236.03,E2 -15236.03} C_VEL
LIN {X 0,Y 322.707,Z 172.494,A -85,B 0,C 180,E1 -15238.627,E2 -15238.627} C_VEL
LIN {X 0,Y 319.999,Z 160.573,A -85,B 0,C 180,E1 -15242.179,E2 -15242.179} C_VEL
LIN {X 0,Y 319.585,Z 158.676,A -85,B 0,C 180,E1 -15242.777,E2 -15242.777} C_VEL
LIN {X 0,Y 319.552,Z 158.675,A -85,B 0,C 180,E1 -15246.427,E2 -15246.427} C_VEL
LIN {X 0,Y 319.524,Z 158.683,A -85,B 0,C 180,E1 -15249.661,E2 -15249.661} C_VEL
LIN {X 0,Y 319.515,Z 158.686,A -85,B 0,C 180,E1 -15253.459,E2 -15253.459} C_VEL
LIN {X 0,Y 319.546,Z 158.682,A -85,B 0,C 180,E1 -15257.015,E2 -15257.015} C_VEL
LIN {X 0,Y 319.539,Z 158.679,A -85,B 0,C 180,E1 -15260.37,E2 -15260.37} C_VEL
LIN {X 0,Y 319.572,Z 158.676,A -85,B 0,C 180,E1 -15264.457,E2 -15264.457} C_VEL
LIN {X 0,Y 319.517,Z 158.681,A -85,B 0,C 180,E1 -15268.136,E2 -15268.136} C_VEL
LIN {X 0,Y 319.563,Z 158.672,A -85,B 0,C 180,E1 -15271.603,E2 -15271.603} C_VEL
LIN {X 0,Y 319.519,Z 158.681,A -85,B 0,C 180,E1 -15275.297,E2 -15275.297} C_VEL
LIN {X 0,Y 319.554,Z 158.675,A -85,B 0,C 180,E1 -15278.045,E2 -15278.045} C_VEL
LIN {X 0,Y 319.578,Z 158.676,A -85,B 0,C 180,E1 -15282.068,E2 -15282.068} C_VEL
LIN {X 0,Y 319.7,Z 158.661,A -85,B 0,C 180,E1 -15286.006,E2 -15286.006} C_VEL
LIN {X 0,Y 319.725,Z 158.656,A -85,B 0,C 180,E1 -15289.872,E2 -15289.872} C_VEL
LIN {X 0,Y 319.887,Z 158.637,A -85,B 0,C 180,E1 -15293.693,E2 -15293.693} C_VEL
LIN {X 0,Y 319.938,Z 158.626,A -85,B 0,C 180,E1 -15297.482,E2 -15297.482} C_VEL
LIN {X 0,Y 319.988,Z 158.624,A -85,B 0,C 180,E1 -15301.259,E2 -15301.259} C_VEL
LIN {X 0,Y 319.691,Z 158.661,A -85,B 0,C 180,E1 -15303.782,E2 -15303.782} C_VEL
LIN {X 0,Y 319.879,Z 158.636,A -85,B 0,C 180,E1 -15306.431,E2 -15306.431} C_VEL
LIN {X 0,Y 319.727,Z 158.656,A -85,B 0,C 180,E1 -15310.128,E2 -15310.128} C_VEL
LIN {X 0,Y 319.701,Z 158.66,A -85,B 0,C 180,E1 -15313.994,E2 -15313.994} C_VEL
LIN {X 0,Y 319.579,Z 158.673,A -85,B 0,C 180,E1 -15317.932,E2 -15317.932} C_VEL
LIN {X 0,Y 319.58,Z 158.675,A -85,B 0,C 180,E1 -15321.954,E2 -15321.954} C_VEL
LIN {X 0,Y 319.545,Z 158.675,A -85,B 0,C 180,E1 -15326.096,E2 -15326.096} C_VEL
LIN {X 0,Y 319.536,Z 158.683,A -85,B 0,C 180,E1 -15328.939,E2 -15328.939} C_VEL
LIN {X 0,Y 319.517,Z 158.68,A -85,B 0,C 180,E1 -15331.864,E2 -15331.864} C_VEL
LIN {X 0,Y 319.572,Z 158.676,A -85,B 0,C 180,E1 -15335.543,E2 -15335.543} C_VEL
LIN {X 0,Y 319.523,Z 158.681,A -85,B 0,C 180,E1 -15339.663,E2 -15339.663} C_VEL
LIN {X 0,Y 319.515,Z 158.682,A -85,B 0,C 180,E1 -15343.461,E2 -15343.461} C_VEL
LIN {X 0,Y 319.549,Z 158.68,A -85,B 0,C 180,E1 -15347.017,E2 -15347.017} C_VEL
LIN {X 0,Y 319.541,Z 158.683,A -85,B 0,C 180,E1 -15350.372,E2 -15350.372} C_VEL
LIN {X 0,Y 319.577,Z 158.678,A -85,B 0,C 180,E1 -15354.458,E2 -15354.458} C_VEL
LIN {X 0,Y 319.522,Z 158.686,A -85,B 0,C 180,E1 -15358.138,E2 -15358.138} C_VEL
LIN {X 0,Y 319.57,Z 158.675,A -85,B 0,C 180,E1 -15361.605,E2 -15361.605} C_VEL
LIN {X 0,Y 319.594,Z 158.676,A -85,B 0,C 180,E1 -15362.853,E2 -15362.853} C_VEL
LIN {X 0,Y 320.946,Z 164.665,A -85,B 0,C 180,E1 -15364.775,E2 -15364.775} C_VEL
LIN {X 0,Y 329.797,Z 186.865,A -85,B 0,C 180,E1 -15366.034,E2 -15366.034} C_VEL
LIN {X 0,Y 331.245,Z 194.846,A -85,B 0,C 180,E1 -15366.332,E2 -15366.332} C_VEL
LIN {X 0,Y 329.702,Z 266.987,A -85,B 0,C 180,E1 -15367.892,E2 -15367.892} C_VEL
LIN {X 0,Y 329.192,Z 279.833,A -85,B 0,C 180,E1 -15368.31,E2 -15368.31} C_VEL
LIN {X 0,Y 328.315,Z 293.049,A -85,B 0,C 180,E1 -15368.99,E2 -15368.99} C_VEL
LIN {X 0,Y 327.246,Z 305.415,A -85,B 0,C 180,E1 -15369.904,E2 -15369.904} C_VEL
LIN {X 0,Y 326.003,Z 316.502,A -85,B 0,C 180,E1 -15370.971,E2 -15370.971} C_VEL
LIN {X 0,Y 324.752,Z 327.791,A -85,B 0,C 180,E1 -15372.365,E2 -15372.365} C_VEL
LIN {X 0,Y 323.377,Z 337.751,A -85,B 0,C 180,E1 -15373.914,E2 -15373.914} C_VEL
LIN {X 0,Y 321.897,Z 347.383,A -85,B 0,C 180,E1 -15375.782,E2 -15375.782} C_VEL
LIN {X 0,Y 320.681,Z 355.061,A -85,B 0,C 180,E1 -15377.663,E2 -15377.663} C_VEL
LIN {X 0,Y 319.882,Z 360.299,A -85,B 0,C 180,E1 -15379.238,E2 -15379.238} C_VEL
LIN {X 0,Y 319.119,Z 365.38,A -85,B 0,C 180,E1 -15381.133,E2 -15381.133} C_VEL
LIN {X 0,Y 318.588,Z 369.39,A -85,B 0,C 180,E1 -15383.071,E2 -15383.071} C_VEL
LIN {X 0,Y 318.292,Z 372.232,A -85,B 0,C 180,E1 -15384.934,E2 -15384.934} C_VEL
LIN {X 0,Y 318.065,Z 373.628,A -85,B 0,C 180,E1 -15386.2,E2 -15386.2} C_VEL
LIN {X 0,Y 317.859,Z 375.231,A -85,B 0,C 180,E1 -15388.734,E2 -15388.734} C_VEL
LIN {X 0,Y 317.861,Z 375.461,A -85,B 0,C 180,E1 -15390.001,E2 -15390.001} C_VEL
LIN {X 0,Y 317.859,Z 375.271,A -85,B 0,C 180,E1 -15391.268,E2 -15391.268} C_VEL
LIN {X 0,Y 318.061,Z 373.721,A -85,B 0,C 180,E1 -15393.801,E2 -15393.801} C_VEL
LIN {X 0,Y 318.264,Z 372.366,A -85,B 0,C 180,E1 -15395.068,E2 -15395.068} C_VEL
LIN {X 0,Y 318.633,Z 369.462,A -85,B 0,C 180,E1 -15396.994,E2 -15396.994} C_VEL
LIN {X 0,Y 319.036,Z 365.629,A -85,B 0,C 180,E1 -15398.871,E2 -15398.871} C_VEL
LIN {X 0,Y 319.846,Z 360.618,A -85,B 0,C 180,E1 -15400.765,E2 -15400.765} C_VEL
LIN {X 0,Y 320.828,Z 354.31,A -85,B 0,C 180,E1 -15402.654,E2 -15402.654} C_VEL
LIN {X 0,Y 322.05,Z 346.412,A -85,B 0,C 180,E1 -15404.535,E2 -15404.535} C_VEL
LIN {X 0,Y 323.634,Z 336.58,A -85,B 0,C 180,E1 -15406.398,E2 -15406.398} C_VEL
LIN {X 0,Y 324.858,Z 327.082,A -85,B 0,C 180,E1 -15407.842,E2 -15407.842} C_VEL
LIN {X 0,Y 326.161,Z 316.042,A -85,B 0,C 180,E1 -15409.184,E2 -15409.184} C_VEL
LIN {X 0,Y 327.374,Z 304.85,A -85,B 0,C 180,E1 -15410.254,E2 -15410.254} C_VEL
LIN {X 0,Y 328.481,Z 292.229,A -85,B 0,C 180,E1 -15411.165,E2 -15411.165} C_VEL
LIN {X 0,Y 329.238,Z 279.573,A -85,B 0,C 180,E1 -15411.812,E2 -15411.812} C_VEL
LIN {X 0,Y 329.853,Z 266.539,A -85,B 0,C 180,E1 -15412.222,E2 -15412.222} C_VEL
LIN {X 0,Y 331.319,Z 194.285,A -85,B 0,C 180,E1 -15413.789,E2 -15413.789} C_VEL
LIN {X 0,Y 329.379,Z 185.816,A -85,B 0,C 180,E1 -15414.138,E2 -15414.138} C_VEL
LIN {X 0,Y 321.729,Z 166.75,A -85,B 0,C 180,E1 -15415.217,E2 -15415.217} C_VEL
LIN {X 0,Y 320.926,Z 164.536,A -85,B 0,C 180,E1 -15415.382,E2 -15415.382} C_VEL
LIN {X 0,Y 319.614,Z 158.674,A -85,B 0,C 180,E1 -15417.324,E2 -15417.324} C_VEL
LIN {X 0,Y 319.552,Z 158.679,A -85,B 0,C 180,E1 -15420.936,E2 -15420.936} C_VEL
LIN {X 0,Y 319.522,Z 158.68,A -85,B 0,C 180,E1 -15422.331,E2 -15422.331} C_VEL
LIN {X 0,Y 318.874,Z 158.765,A -85,B 0,C 180,E1 -15423.384,E2 -15423.384} C_VEL
LIN {X 0,Y 316.042,Z 159.116,A -85,B 0,C 180,E1 -15425.099,E2 -15425.099} C_VEL
LIN {X 0,Y 313.623,Z 159.417,A -85,B 0,C 180,E1 -15426.488,E2 -15426.488} C_VEL
LIN {X 0,Y 312.573,Z 159.551,A -85,B 0,C 180,E1 -15427.564,E2 -15427.564} C_VEL
LIN {X 0,Y 312.481,Z 159.56,A -85,B 0,C 180,E1 -15427.929,E2 -15427.929} C_VEL
LIN {X 0,Y 312.456,Z 159.563,A -85,B 0,C 180,E1 -15432.075,E2 -15432.075} C_VEL
LIN {X 0,Y 312.458,Z 159.56,A -85,B 0,C 180,E1 -15436.035,E2 -15436.035} C_VEL
LIN {X 0,Y 312.455,Z 159.559,A -85,B 0,C 180,E1 -15439.885,E2 -15439.885} C_VEL
LIN {X 0,Y 312.533,Z 159.55,A -85,B 0,C 180,E1 -15444.051,E2 -15444.051} C_VEL
LIN {X 0,Y 312.501,Z 159.559,A -85,B 0,C 180,E1 -15447.333,E2 -15447.333} C_VEL
LIN {X 0,Y 312.506,Z 159.555,A -85,B 0,C 180,E1 -15451.292,E2 -15451.292} C_VEL
LIN {X 0,Y 312.547,Z 159.555,A -85,B 0,C 180,E1 -15454.707,E2 -15454.707} C_VEL
LIN {X 0,Y 312.582,Z 159.54,A -85,B 0,C 180,E1 -15457.528,E2 -15457.528} C_VEL
LIN {X 0,Y 312.55,Z 159.55,A -85,B 0,C 180,E1 -15461.651,E2 -15461.651} C_VEL
LIN {X 0,Y 312.65,Z 159.532,A -85,B 0,C 180,E1 -15465.684,E2 -15465.684} C_VEL
LIN {X 0,Y 312.684,Z 159.534,A -85,B 0,C 180,E1 -15469.641,E2 -15469.641} C_VEL
LIN {X 0,Y 312.794,Z 159.517,A -85,B 0,C 180,E1 -15472.252,E2 -15472.252} C_VEL
LIN {X 0,Y 312.682,Z 159.533,A -85,B 0,C 180,E1 -15474.842,E2 -15474.842} C_VEL
LIN {X 0,Y 312.964,Z 159.497,A -85,B 0,C 180,E1 -15478.713,E2 -15478.713} C_VEL
LIN {X 0,Y 312.963,Z 159.491,A -85,B 0,C 180,E1 -15481.287,E2 -15481.287} C_VEL
LIN {X 0,Y 312.837,Z 159.514,A -85,B 0,C 180,E1 -15486.449,E2 -15486.449} C_VEL
LIN {X 0,Y 312.679,Z 159.531,A -85,B 0,C 180,E1 -15490.359,E2 -15490.359} C_VEL
LIN {X 0,Y 312.602,Z 159.542,A -85,B 0,C 180,E1 -15494.82,E2 -15494.82} C_VEL
LIN {X 0,Y 312.531,Z 159.553,A -85,B 0,C 180,E1 -15499.184,E2 -15499.184} C_VEL
LIN {X 0,Y 312.512,Z 159.552,A -85,B 0,C 180,E1 -15502.775,E2 -15502.775} C_VEL
LIN {X 0,Y 312.481,Z 159.56,A -85,B 0,C 180,E1 -15506.732,E2 -15506.732} C_VEL
LIN {X 0,Y 312.493,Z 159.558,A -85,B 0,C 180,E1 -15509.655,E2 -15509.655} C_VEL
LIN {X 0,Y 312.519,Z 159.552,A -85,B 0,C 180,E1 -15513.689,E2 -15513.689} C_VEL
LIN {X 0,Y 312.513,Z 159.554,A -85,B 0,C 180,E1 -15517.387,E2 -15517.387} C_VEL
LIN {X 0,Y 312.44,Z 159.568,A -85,B 0,C 180,E1 -15520.717,E2 -15520.717} C_VEL
LIN {X 0,Y 312.45,Z 159.563,A -85,B 0,C 180,E1 -15524.21,E2 -15524.21} C_VEL
LIN {X 0,Y 312.454,Z 159.562,A -85,B 0,C 180,E1 -15527.925,E2 -15527.925} C_VEL
LIN {X 0,Y 312.484,Z 159.558,A -85,B 0,C 180,E1 -15531.923,E2 -15531.923} C_VEL
LIN {X 0,Y 312.532,Z 159.556,A -85,B 0,C 180,E1 -15534.22,E2 -15534.22} C_VEL
LIN {X 0,Y 312.553,Z 159.618,A -85,B 0,C 180,E1 -15536.737,E2 -15536.737} C_VEL
LIN {X 0,Y 315.232,Z 171.474,A -85,B 0,C 180,E1 -15540.4,E2 -15540.4} C_VEL
LIN {X 0,Y 317.213,Z 181.726,A -85,B 0,C 180,E1 -15543.399,E2 -15543.399} C_VEL
LIN {X 0,Y 317.175,Z 185.341,A -85,B 0,C 180,E1 -15544.375,E2 -15544.375} C_VEL
LIN {X 0,Y 322.095,Z 213.602,A -85,B 0,C 180,E1 -15545.473,E2 -15545.473} C_VEL
LIN {X 0,Y 324.093,Z 227.521,A -85,B 0,C 180,E1 -15545.963,E2 -15545.963} C_VEL
LIN {X 0,Y 322.577,Z 294.194,A -85,B 0,C 180,E1 -15547.46,E2 -15547.46} C_VEL
LIN {X 0,Y 321.738,Z 307.374,A -85,B 0,C 180,E1 -15547.99,E2 -15547.99} C_VEL
LIN {X 0,Y 320.61,Z 319.488,A -85,B 0,C 180,E1 -15548.711,E2 -15548.711} C_VEL
LIN {X 0,Y 319.225,Z 331.721,A -85,B 0,C 180,E1 -15549.711,E2 -15549.711} C_VEL
LIN {X 0,Y 317.717,Z 343.306,A -85,B 0,C 180,E1 -15550.957,E2 -15550.957} C_VEL
LIN {X 0,Y 316.15,Z 353.739,A -85,B 0,C 180,E1 -15552.369,E2 -15552.369} C_VEL
LIN {X 0,Y 314.86,Z 363.462,A -85,B 0,C 180,E1 -15554.03,E2 -15554.03} C_VEL
LIN {X 0,Y 313.595,Z 371.54,A -85,B 0,C 180,E1 -15555.728,E2 -15555.728} C_VEL
LIN {X 0,Y 312.392,Z 378.981,A -85,B 0,C 180,E1 -15557.659,E2 -15557.659} C_VEL
LIN {X 0,Y 311.619,Z 384.966,A -85,B 0,C 180,E1 -15559.605,E2 -15559.605} C_VEL
LIN {X 0,Y 311.116,Z 389.699,A -85,B 0,C 180,E1 -15561.556,E2 -15561.556} C_VEL
LIN {X 0,Y 310.811,Z 393.318,A -85,B 0,C 180,E1 -15563.508,E2 -15563.508} C_VEL
LIN {X 0,Y 310.706,Z 395.185,A -85,B 0,C 180,E1 -15564.808,E2 -15564.808} C_VEL
LIN {X 0,Y 310.716,Z 396.588,A -85,B 0,C 180,E1 -15566.109,E2 -15566.109} C_VEL
LIN {X 0,Y 310.701,Z 397.589,A -85,B 0,C 180,E1 -15567.406,E2 -15567.406} C_VEL
LIN {X 0,Y 310.7,Z 398.199,A -85,B 0,C 180,E1 -15568.703,E2 -15568.703} C_VEL
LIN {X 0,Y 310.758,Z 398.415,A -85,B 0,C 180,E1 -15569.999,E2 -15569.999} C_VEL
LIN {X 0,Y 310.7,Z 398.192,A -85,B 0,C 180,E1 -15571.295,E2 -15571.295} C_VEL
LIN {X 0,Y 310.701,Z 397.578,A -85,B 0,C 180,E1 -15572.592,E2 -15572.592} C_VEL
LIN {X 0,Y 310.717,Z 396.574,A -85,B 0,C 180,E1 -15573.89,E2 -15573.89} C_VEL
LIN {X 0,Y 310.731,Z 394.562,A -85,B 0,C 180,E1 -15575.628,E2 -15575.628} C_VEL
LIN {X 0,Y 311.004,Z 390.976,A -85,B 0,C 180,E1 -15577.792,E2 -15577.792} C_VEL
LIN {X 0,Y 311.414,Z 386.613,A -85,B 0,C 180,E1 -15579.744,E2 -15579.744} C_VEL
LIN {X 0,Y 312.077,Z 381.062,A -85,B 0,C 180,E1 -15581.693,E2 -15581.693} C_VEL
LIN {X 0,Y 313.169,Z 374.144,A -85,B 0,C 180,E1 -15583.628,E2 -15583.628} C_VEL
LIN {X 0,Y 314.521,Z 365.489,A -85,B 0,C 180,E1 -15585.553,E2 -15585.553} C_VEL
LIN {X 0,Y 315.733,Z 356.614,A -85,B 0,C 180,E1 -15587.153,E2 -15587.153} C_VEL
LIN {X 0,Y 317.323,Z 345.701,A -85,B 0,C 180,E1 -15588.731,E2 -15588.731} C_VEL
LIN {X 0,Y 318.824,Z 334.686,A -85,B 0,C 180,E1 -15589.978,E2 -15589.978} C_VEL
LIN {X 0,Y 320.259,Z 322.34,A -85,B 0,C 180,E1 -15591.059,E2 -15591.059} C_VEL
LIN {X 0,Y 321.383,Z 310.646,A -85,B 0,C 180,E1 -15591.823,E2 -15591.823} C_VEL
LIN {X 0,Y 322.346,Z 298.143,A -85,B 0,C 180,E1 -15592.386,E2 -15592.386} C_VEL
LIN {X 0,Y 322.878,Z 282.188,A -85,B 0,C 180,E1 -15592.812,E2 -15592.812} C_VEL
LIN {X 0,Y 323.94,Z 226.457,A -85,B 0,C 180,E1 -15594.05,E2 -15594.05} C_VEL
LIN {X 0,Y 319.871,Z 200.515,A -85,B 0,C 180,E1 -15594.998,E2 -15594.998} C_VEL
LIN {X 0,Y 317.15,Z 185.257,A -85,B 0,C 180,E1 -15595.624,E2 -15595.624} C_VEL
LIN {X 0,Y 317.166,Z 181.635,A -85,B 0,C 180,E1 -15596.603,E2 -15596.603} C_VEL
LIN {X 0,Y 315.381,Z 172.195,A -85,B 0,C 180,E1 -15599.356,E2 -15599.356} C_VEL
LIN {X 0,Y 312.706,Z 160.406,A -85,B 0,C 180,E1 -15602.984,E2 -15602.984} C_VEL
LIN {X 0,Y 312.529,Z 159.555,A -85,B 0,C 180,E1 -15603.264,E2 -15603.264} C_VEL
LIN {X 0,Y 312.531,Z 159.55,A -85,B 0,C 180,E1 -15605.948,E2 -15605.948} C_VEL
LIN {X 0,Y 312.451,Z 159.561,A -85,B 0,C 180,E1 -15610.114,E2 -15610.114} C_VEL
LIN {X 0,Y 312.452,Z 159.563,A -85,B 0,C 180,E1 -15613.964,E2 -15613.964} C_VEL
LIN {X 0,Y 312.449,Z 159.563,A -85,B 0,C 180,E1 -15617.924,E2 -15617.924} C_VEL
LIN {X 0,Y 312.477,Z 159.559,A -85,B 0,C 180,E1 -15621.922,E2 -15621.922} C_VEL
LIN {X 0,Y 312.523,Z 159.553,A -85,B 0,C 180,E1 -15624.219,E2 -15624.219} C_VEL
LIN {X 0,Y 312.495,Z 159.556,A -85,B 0,C 180,E1 -15627.333,E2 -15627.333} C_VEL
LIN {X 0,Y 312.498,Z 159.553,A -85,B 0,C 180,E1 -15631.291,E2 -15631.291} C_VEL
LIN {X 0,Y 312.51,Z 159.559,A -85,B 0,C 180,E1 -15634.704,E2 -15634.704} C_VEL
LIN {X 0,Y 312.531,Z 159.548,A -85,B 0,C 180,E1 -15637.525,E2 -15637.525} C_VEL
LIN {X 0,Y 312.538,Z 159.551,A -85,B 0,C 180,E1 -15641.65,E2 -15641.65} C_VEL
LIN {X 0,Y 312.643,Z 159.538,A -85,B 0,C 180,E1 -15645.684,E2 -15645.684} C_VEL
LIN {X 0,Y 312.675,Z 159.532,A -85,B 0,C 180,E1 -15649.641,E2 -15649.641} C_VEL
LIN {X 0,Y 312.829,Z 159.516,A -85,B 0,C 180,E1 -15653.55,E2 -15653.55} C_VEL
LIN {X 0,Y 312.956,Z 159.497,A -85,B 0,C 180,E1 -15658.713,E2 -15658.713} C_VEL
LIN {X 0,Y 312.957,Z 159.5,A -85,B 0,C 180,E1 -15661.287,E2 -15661.287} C_VEL
LIN {X 0,Y 312.678,Z 159.528,A -85,B 0,C 180,E1 -15665.158,E2 -15665.158} C_VEL
LIN {X 0,Y 312.788,Z 159.524,A -85,B 0,C 180,E1 -15667.748,E2 -15667.748} C_VEL
LIN {X 0,Y 312.653,Z 159.536,A -85,B 0,C 180,E1 -15671.672,E2 -15671.672} C_VEL
LIN {X 0,Y 312.606,Z 159.542,A -85,B 0,C 180,E1 -15674.828,E2 -15674.828} C_VEL
LIN {X 0,Y 312.538,Z 159.551,A -85,B 0,C 180,E1 -15679.192,E2 -15679.192} C_VEL
LIN {X 0,Y 312.525,Z 159.554,A -85,B 0,C 180,E1 -15682.784,E2 -15682.784} C_VEL
LIN {X 0,Y 312.479,Z 159.556,A -85,B 0,C 180,E1 -15686.732,E2 -15686.732} C_VEL
LIN {X 0,Y 312.489,Z 159.558,A -85,B 0,C 180,E1 -15689.656,E2 -15689.656} C_VEL
LIN {X 0,Y 312.513,Z 159.555,A -85,B 0,C 180,E1 -15693.69,E2 -15693.69} C_VEL
LIN {X 0,Y 312.507,Z 159.556,A -85,B 0,C 180,E1 -15697.388,E2 -15697.388} C_VEL
LIN {X 0,Y 312.435,Z 159.568,A -85,B 0,C 180,E1 -15700.718,E2 -15700.718} C_VEL
LIN {X 0,Y 312.446,Z 159.564,A -85,B 0,C 180,E1 -15704.211,E2 -15704.211} C_VEL
LIN {X 0,Y 312.463,Z 159.561,A -85,B 0,C 180,E1 -15707.923,E2 -15707.923} C_VEL
LIN {X 0,Y 312.491,Z 159.558,A -85,B 0,C 180,E1 -15710.972,E2 -15710.972} C_VEL
LIN {X 0,Y 312.529,Z 159.556,A -85,B 0,C 180,E1 -15714.221,E2 -15714.221} C_VEL
LIN {X 0,Y 312.499,Z 159.557,A -85,B 0,C 180,E1 -15717.335,E2 -15717.335} C_VEL
LIN {X 0,Y 312.505,Z 159.554,A -85,B 0,C 180,E1 -15721.293,E2 -15721.293} C_VEL
LIN {X 0,Y 312.528,Z 159.68,A -85,B 0,C 180,E1 -15722.414,E2 -15722.414} C_VEL
LIN {X 0,Y 313.778,Z 165.079,A -85,B 0,C 180,E1 -15724.166,E2 -15724.166} C_VEL
LIN {X 0,Y 321.83,Z 184.594,A -85,B 0,C 180,E1 -15725.338,E2 -15725.338} C_VEL
LIN {X 0,Y 323.885,Z 190.679,A -85,B 0,C 180,E1 -15725.653,E2 -15725.653} C_VEL
LIN {X 0,Y 324.75,Z 195.16,A -85,B 0,C 180,E1 -15725.83,E2 -15725.83} C_VEL
LIN {X 0,Y 322.989,Z 271.707,A -85,B 0,C 180,E1 -15727.534,E2 -15727.534} C_VEL
LIN {X 0,Y 322.349,Z 285.095,A -85,B 0,C 180,E1 -15728.078,E2 -15728.078} C_VEL
LIN {X 0,Y 321.572,Z 295.599,A -85,B 0,C 180,E1 -15728.695,E2 -15728.695} C_VEL
LIN {X 0,Y 320.394,Z 307.443,A -85,B 0,C 180,E1 -15729.622,E2 -15729.622} C_VEL
LIN {X 0,Y 319.149,Z 318.186,A -85,B 0,C 180,E1 -15730.713,E2 -15730.713} C_VEL
LIN {X 0,Y 317.986,Z 328.054,A -85,B 0,C 180,E1 -15731.977,E2 -15731.977} C_VEL
LIN {X 0,Y 316.581,Z 338.013,A -85,B 0,C 180,E1 -15733.559,E2 -15733.559} C_VEL
LIN {X 0,Y 315.026,Z 347.644,A -85,B 0,C 180,E1 -15735.465,E2 -15735.465} C_VEL
LIN {X 0,Y 313.754,Z 355.322,A -85,B 0,C 180,E1 -15737.386,E2 -15737.386} C_VEL
LIN {X 0,Y 312.913,Z 360.56,A -85,B 0,C 180,E1 -15738.995,E2 -15738.995} C_VEL
LIN {X 0,Y 312.088,Z 365.641,A -85,B 0,C 180,E1 -15740.931,E2 -15740.931} C_VEL
LIN {X 0,Y 311.491,Z 369.951,A -85,B 0,C 180,E1 -15743.098,E2 -15743.098} C_VEL
LIN {X 0,Y 311.22,Z 372.492,A -85,B 0,C 180,E1 -15744.818,E2 -15744.818} C_VEL
LIN {X 0,Y 311.002,Z 373.887,A -85,B 0,C 180,E1 -15746.113,E2 -15746.113} C_VEL
LIN {X 0,Y 310.77,Z 375.49,A -85,B 0,C 180,E1 -15748.705,E2 -15748.705} C_VEL
LIN {X 0,Y 310.768,Z 375.72,A -85,B 0,C 180,E1 -15750.001,E2 -15750.001} C_VEL
LIN {X 0,Y 310.77,Z 375.53,A -85,B 0,C 180,E1 -15751.297,E2 -15751.297} C_VEL
LIN {X 0,Y 310.997,Z 373.979,A -85,B 0,C 180,E1 -15753.888,E2 -15753.888} C_VEL
LIN {X 0,Y 311.194,Z 372.624,A -85,B 0,C 180,E1 -15755.184,E2 -15755.184} C_VEL
LIN {X 0,Y 311.554,Z 369.975,A -85,B 0,C 180,E1 -15756.996,E2 -15756.996} C_VEL
LIN {X 0,Y 312.01,Z 365.887,A -85,B 0,C 180,E1 -15759.072,E2 -15759.072} C_VEL
LIN {X 0,Y 312.878,Z 360.876,A -85,B 0,C 180,E1 -15761.008,E2 -15761.008} C_VEL
LIN {X 0,Y 313.904,Z 354.567,A -85,B 0,C 180,E1 -15762.938,E2 -15762.938} C_VEL
LIN {X 0,Y 315.18,Z 346.669,A -85,B 0,C 180,E1 -15764.859,E2 -15764.859} C_VEL
LIN {X 0,Y 316.83,Z 336.836,A -85,B 0,C 180,E1 -15766.761,E2 -15766.761} C_VEL
LIN {X 0,Y 318.186,Z 326.524,A -85,B 0,C 180,E1 -15768.345,E2 -15768.345} C_VEL
LIN {X 0,Y 319.488,Z 316.295,A -85,B 0,C 180,E1 -15769.601,E2 -15769.601} C_VEL
LIN {X 0,Y 320.752,Z 305.102,A -85,B 0,C 180,E1 -15770.691,E2 -15770.691} C_VEL
LIN {X 0,Y 321.887,Z 292.479,A -85,B 0,C 180,E1 -15771.62,E2 -15771.62} C_VEL
LIN {X 0,Y 322.681,Z 279.819,A -85,B 0,C 180,E1 -15772.279,E2 -15772.279} C_VEL
LIN {X 0,Y 323.311,Z 266.776,A -85,B 0,C 180,E1 -15772.696,E2 -15772.696} C_VEL
LIN {X 0,Y 324.729,Z 194.785,A -85,B 0,C 180,E1 -15774.296,E2 -15774.296} C_VEL
LIN {X 0,Y 323.176,Z 188.166,A -85,B 0,C 180,E1 -15774.58,E2 -15774.58} C_VEL
LIN {X 0,Y 314.996,Z 167.905,A -85,B 0,C 180,E1 -15775.773,E2 -15775.773} C_VEL
LIN {X 0,Y 313.752,Z 164.873,A -85,B 0,C 180,E1 -15775.988,E2 -15775.988} C_VEL
LIN {X 0,Y 312.534,Z 159.556,A -85,B 0,C 180,E1 -15777.815,E2 -15777.815} C_VEL
LIN {X 0,Y 312.504,Z 159.555,A -85,B 0,C 180,E1 -15781.285,E2 -15781.285} C_VEL
LIN {X 0,Y 312.508,Z 159.556,A -85,B 0,C 180,E1 -15784.21,E2 -15784.21} C_VEL
LIN {X 0,Y 312.512,Z 159.557,A -85,B 0,C 180,E1 -15787.387,E2 -15787.387} C_VEL
